C03656=1201.315,301.824,-68.864,-176.578,7.338,148.389
C03657=1201.311,302.072,-68.893,-176.576,7.341,148.389
C03658=1201.307,302.320,-68.924,-176.573,7.344,148.389
C03659=1201.303,302.568,-68.953,-176.571,7.347,148.389
C03660=1201.298,302.817,-68.983,-176.568,7.350,148.389
C03661=1201.294,303.064,-69.013,-176.566,7.352,148.389
C03662=1201.290,303.313,-69.043,-176.563,7.355,148.389
C03663=1201.285,303.561,-69.073,-176.561,7.358,148.389
C03664=1201.281,303.809,-69.103,-176.559,7.360,148.388
C03665=1201.277,304.057,-69.132,-176.556,7.363,148.388
C03666=1201.272,304.306,-69.162,-176.554,7.366,148.389
C03667=1201.268,304.553,-69.193,-176.551,7.369,148.389
C03668=1201.264,304.802,-69.222,-176.549,7.372,148.389
C03669=1201.260,305.050,-69.253,-176.546,7.375,148.389
C03670=1201.255,305.299,-69.283,-176.544,7.377,148.389
C03671=1201.251,305.547,-69.313,-176.541,7.380,148.389
C03672=1201.247,305.795,-69.343,-176.539,7.382,148.388
C03673=1201.243,306.042,-69.373,-176.536,7.385,148.388
C03674=1201.238,306.291,-69.403,-176.534,7.388,148.388
C03675=1201.234,306.539,-69.433,-176.532,7.390,148.388
C03676=1201.229,306.787,-69.463,-176.529,7.393,148.388
C03677=1201.225,307.035,-69.493,-176.527,7.397,148.389
C03678=1201.220,307.283,-69.524,-176.525,7.399,148.388
C03679=1201.217,307.532,-69.554,-176.522,7.402,148.388
C03680=1201.213,307.780,-69.584,-176.519,7.405,148.388
C03681=1201.208,308.028,-69.614,-176.517,7.407,148.388
C03682=1201.204,308.276,-69.644,-176.514,7.410,148.388
C03683=1201.199,308.524,-69.675,-176.512,7.413,148.388
C03684=1201.196,308.772,-69.705,-176.510,7.416,148.389
C03685=1201.191,309.020,-69.735,-176.507,7.419,148.389
C03686=1201.187,309.269,-69.765,-176.505,7.422,148.389
C03687=1201.183,309.517,-69.796,-176.502,7.424,148.388
C03688=1201.179,309.764,-69.826,-176.500,7.427,148.388
C03689=1201.174,310.013,-69.856,-176.497,7.430,148.388
C03690=1201.170,310.261,-69.886,-176.495,7.432,148.388
C03691=1201.165,310.509,-69.917,-176.493,7.435,148.389
C03692=1201.161,310.758,-69.948,-176.490,7.439,148.389
C03693=1201.157,311.006,-69.978,-176.488,7.441,148.389
C03694=1201.153,311.253,-70.009,-176.485,7.444,148.389
C03695=1201.149,311.501,-70.039,-176.483,7.447,148.389
C03696=1201.144,311.749,-70.069,-176.481,7.449,148.389
C03697=1201.141,311.998,-70.099,-176.478,7.452,148.389
C03698=1201.136,312.246,-70.130,-176.475,7.455,148.389
C03699=1201.131,312.494,-70.161,-176.473,7.457,148.389
C03700=1201.127,312.742,-70.191,-176.471,7.461,148.389
C03701=1201.123,312.990,-70.222,-176.468,7.464,148.389
C03702=1201.119,313.239,-70.252,-176.466,7.466,148.389
C03703=1201.115,313.487,-70.282,-176.464,7.469,148.389
C03704=1201.110,313.734,-70.313,-176.461,7.472,148.389
C03705=1201.105,313.982,-70.344,-176.459,7.474,148.389
C03706=1201.102,314.231,-70.374,-176.457,7.478,148.389
C03707=1201.097,314.507,-70.409,-176.454,7.481,148.389
C03708=1201.092,314.783,-70.442,-176.451,7.484,148.389
C03709=1201.088,315.059,-70.476,-176.448,7.487,148.389
C03710=1201.083,315.335,-70.511,-176.446,7.490,148.389
C03711=1201.078,315.584,-70.541,-176.444,7.493,148.389
C03712=1201.074,315.832,-70.572,-176.441,7.496,148.389
C03713=1201.071,316.080,-70.602,-176.439,7.498,148.389
C03714=1201.066,316.328,-70.633,-176.436,7.501,148.389
C03715=1201.062,316.575,-70.665,-176.434,7.505,148.389
C03716=1201.058,316.824,-70.696,-176.432,7.507,148.389
C03717=1201.054,317.072,-70.726,-176.429,7.510,148.389
C03718=1201.049,317.320,-70.757,-176.426,7.513,148.389
C03719=1201.044,317.568,-70.788,-176.425,7.515,148.389
C03720=1201.040,317.816,-70.819,-176.422,7.518,148.389
C03721=1201.037,318.064,-70.849,-176.419,7.521,148.389
C03722=1201.032,318.312,-70.880,-176.417,7.525,148.390
C03723=1201.028,318.561,-70.911,-176.415,7.527,148.389
C03724=1201.023,318.809,-70.942,-176.412,7.530,148.389
C03725=1201.019,319.057,-70.972,-176.410,7.533,148.390
C03726=1201.016,319.304,-71.004,-176.408,7.536,148.390
C03727=1201.011,319.552,-71.034,-176.405,7.539,148.390
C03728=1201.007,319.801,-71.065,-176.403,7.542,148.390
C03729=1201.003,320.049,-71.096,-176.401,7.544,148.390
C03730=1200.998,320.297,-71.127,-176.398,7.547,148.390
C03731=1200.994,320.545,-71.159,-176.396,7.550,148.390
C03732=1200.990,320.792,-71.189,-176.394,7.553,148.390
C03733=1200.986,321.040,-71.220,-176.391,7.556,148.390
C03734=1200.982,321.289,-71.251,-176.389,7.559,148.390
C03735=1200.977,321.536,-71.282,-176.387,7.561,148.390
C03736=1200.973,321.785,-71.313,-176.385,7.565,148.390
C03737=1200.969,322.033,-71.344,-176.382,7.568,148.390
C03738=1200.964,322.280,-71.376,-176.379,7.571,148.390
C03739=1200.960,322.529,-71.407,-176.378,7.573,148.390
C03740=1200.956,322.777,-71.438,-176.375,7.576,148.390
C03741=1200.952,323.025,-71.469,-176.372,7.579,148.390
C03742=1200.948,323.273,-71.500,-176.370,7.582,148.391
C03743=1200.944,323.522,-71.531,-176.368,7.585,148.391
C03744=1200.940,323.769,-71.562,-176.366,7.588,148.391
C03745=1200.935,324.017,-71.593,-176.363,7.590,148.391
C03746=1200.932,324.265,-71.625,-176.361,7.594,148.391
C03747=1200.927,324.513,-71.656,-176.359,7.597,148.391
C03748=1200.923,324.761,-71.687,-176.356,7.600,148.391
C03749=1200.919,325.009,-71.718,-176.354,7.602,148.391
C03750=1200.915,325.257,-71.749,-176.351,7.605,148.391
C03751=1200.910,325.505,-71.781,-176.349,7.608,148.391
C03752=1200.906,325.753,-71.812,-176.347,7.611,148.391
C03753=1200.902,326.001,-71.843,-176.345,7.614,148.392
C03754=1200.897,326.250,-71.875,-176.342,7.617,148.392
C03755=1200.893,326.497,-71.907,-176.341,7.620,148.392
C03756=1200.889,326.746,-71.938,-176.338,7.623,148.392
C03757=1200.885,326.993,-71.969,-176.336,7.626,148.392
C03758=1200.881,327.242,-72.000,-176.333,7.629,148.392
C03759=1200.876,327.489,-72.032,-176.331,7.631,148.392
C03760=1200.873,327.737,-72.064,-176.329,7.634,148.392
C03761=1200.868,327.985,-72.094,-176.326,7.638,148.392
C03762=1200.864,328.233,-72.126,-176.324,7.640,148.392
C03763=1200.860,328.481,-72.157,-176.322,7.643,148.392
C03764=1200.856,328.729,-72.189,-176.319,7.646,148.392
C03765=1200.851,328.977,-72.221,-176.318,7.649,148.393
C03766=1200.847,329.225,-72.252,-176.315,7.652,148.393
C03767=1200.843,329.473,-72.284,-176.313,7.655,148.393
C03768=1200.839,329.721,-72.315,-176.310,7.658,148.393
C03769=1200.835,329.969,-72.347,-176.308,7.661,148.393
C03770=1200.831,330.217,-72.378,-176.306,7.664,148.393
C03771=1200.826,330.465,-72.410,-176.303,7.667,148.393
C03772=1200.822,330.712,-72.442,-176.302,7.670,148.393
C03773=1200.818,330.961,-72.473,-176.299,7.673,148.393
C03774=1200.814,331.208,-72.505,-176.297,7.676,148.394
C03775=1200.810,331.456,-72.536,-176.294,7.679,148.394
C03776=1200.805,331.704,-72.569,-176.293,7.682,148.394
C03777=1200.801,331.953,-72.600,-176.290,7.685,148.394
C03778=1200.797,332.201,-72.631,-176.288,7.688,148.394
C03779=1200.793,332.448,-72.663,-176.286,7.690,148.394
C03780=1200.789,332.696,-72.695,-176.283,7.693,148.394
C03781=1200.784,332.944,-72.727,-176.281,7.697,148.394
C03782=1200.780,333.192,-72.758,-176.279,7.699,148.395
C03783=1200.776,333.440,-72.790,-176.277,7.702,148.395
C03784=1200.771,333.688,-72.822,-176.275,7.706,148.395
C03785=1200.768,333.936,-72.854,-176.272,7.709,148.395
C03786=1200.764,334.184,-72.886,-176.270,7.711,148.395
C03787=1200.760,334.431,-72.917,-176.268,7.714,148.395
C03788=1200.755,334.680,-72.950,-176.266,7.718,148.395
C03789=1200.751,334.928,-72.981,-176.264,7.720,148.395
C03790=1200.747,335.175,-73.013,-176.261,7.723,148.396
C03791=1200.743,335.424,-73.045,-176.259,7.727,148.396
C03792=1200.738,335.671,-73.077,-176.257,7.729,148.396
C03793=1200.735,335.919,-73.109,-176.255,7.732,148.396
C03794=1200.730,336.167,-73.141,-176.253,7.736,148.396
C03795=1200.726,336.415,-73.173,-176.250,7.739,148.396
C03796=1200.721,336.663,-73.205,-176.248,7.741,148.396
C03797=1200.718,336.911,-73.237,-176.246,7.744,148.397
C03798=1200.714,337.159,-73.269,-176.244,7.748,148.397
C03799=1200.709,337.407,-73.301,-176.242,7.750,148.397
C03800=1200.705,337.655,-73.333,-176.239,7.753,148.397
C03801=1200.702,337.903,-73.364,-176.237,7.757,148.397
C03802=1200.697,338.150,-73.397,-176.235,7.760,148.397
C03803=1200.693,338.398,-73.428,-176.233,7.762,148.397
C03804=1200.688,338.647,-73.461,-176.231,7.766,148.398
C03805=1200.684,338.894,-73.492,-176.228,7.769,148.398
C03806=1200.680,339.142,-73.525,-176.227,7.771,148.398
C03807=1200.676,339.390,-73.557,-176.224,7.775,148.398
C03808=1200.672,339.638,-73.590,-176.222,7.778,148.398
C03809=1200.667,339.886,-73.621,-176.220,7.780,148.398
C03810=1200.663,340.134,-73.654,-176.218,7.784,148.399
C03811=1200.659,340.412,-73.690,-176.216,7.787,148.399
C03812=1200.654,340.690,-73.726,-176.213,7.790,148.399
C03813=1200.650,340.969,-73.762,-176.210,7.794,148.399
C03814=1200.645,341.248,-73.798,-176.208,7.797,148.399
C03815=1200.640,341.495,-73.831,-176.206,7.800,148.400
C03816=1200.637,341.743,-73.863,-176.204,7.803,148.400
C03817=1200.632,341.991,-73.895,-176.202,7.807,148.400
C03818=1200.628,342.239,-73.927,-176.200,7.810,148.400
C03819=1200.624,342.486,-73.960,-176.198,7.812,148.400
C03820=1200.620,342.734,-73.992,-176.196,7.816,148.401
C03821=1200.616,342.983,-74.024,-176.194,7.819,148.401
C03822=1200.611,343.230,-74.057,-176.191,7.821,148.401
C03823=1200.608,343.478,-74.089,-176.189,7.825,148.401
C03824=1200.603,343.726,-74.121,-176.187,7.828,148.401
C03825=1200.599,343.973,-74.154,-176.185,7.831,148.401
C03826=1200.595,344.222,-74.186,-176.183,7.834,148.402
C03827=1200.591,344.470,-74.219,-176.181,7.837,148.402
C03828=1200.587,344.718,-74.251,-176.179,7.841,148.402
C03829=1200.582,344.965,-74.283,-176.177,7.843,148.402
C03830=1200.579,345.213,-74.316,-176.175,7.846,148.402
C03831=1200.574,345.461,-74.348,-176.173,7.850,148.403
C03832=1200.570,345.709,-74.382,-176.171,7.852,148.403
C03833=1200.566,345.957,-74.413,-176.169,7.856,148.403
C03834=1200.562,346.205,-74.447,-176.166,7.859,148.403
C03835=1200.557,346.452,-74.479,-176.165,7.861,148.403
C03836=1200.553,346.700,-74.512,-176.163,7.865,148.404
C03837=1200.549,346.948,-74.544,-176.160,7.868,148.404
C03838=1200.545,347.196,-74.577,-176.159,7.871,148.404
C03839=1200.541,347.444,-74.609,-176.156,7.874,148.404
C03840=1200.537,347.691,-74.642,-176.154,7.877,148.405
C03841=1200.533,347.940,-74.674,-176.152,7.881,148.405
C03842=1200.529,348.188,-74.707,-176.150,7.883,148.405
C03843=1200.524,348.435,-74.740,-176.148,7.886,148.405
C03844=1200.520,348.683,-74.772,-176.146,7.890,148.405
C03845=1200.516,348.930,-74.805,-176.145,7.893,148.406
C03846=1200.512,349.179,-74.838,-176.142,7.896,148.406
C03847=1200.507,349.426,-74.871,-176.140,7.899,148.406
C03848=1200.504,349.674,-74.903,-176.138,7.902,148.406
C03849=1200.500,349.922,-74.936,-176.136,7.905,148.407
C03850=1200.495,350.170,-74.969,-176.134,7.908,148.407
C03851=1200.491,350.418,-75.002,-176.132,7.911,148.407
C03852=1200.487,350.666,-75.035,-176.130,7.914,148.407
C03853=1200.483,350.913,-75.067,-176.128,7.918,148.408
C03854=1200.479,351.160,-75.100,-176.127,7.920,148.408
C03855=1200.475,351.408,-75.133,-176.124,7.924,148.408
C03856=1200.470,351.656,-75.165,-176.122,7.927,148.408
C03857=1200.466,351.904,-75.199,-176.121,7.930,148.409
C03858=1200.462,352.152,-75.232,-176.119,7.933,148.409
C03859=1200.459,352.399,-75.264,-176.117,7.937,148.409
C03860=1200.454,352.648,-75.297,-176.115,7.939,148.409
C03861=1200.450,352.895,-75.330,-176.113,7.942,148.410
C03862=1200.446,353.143,-75.363,-176.110,7.946,148.410
C03863=1200.442,353.391,-75.396,-176.109,7.949,148.410
C03864=1200.438,353.639,-75.429,-176.107,7.952,148.410
C03865=1200.433,353.886,-75.463,-176.105,7.955,148.411
C03866=1200.429,354.135,-75.495,-176.103,7.958,148.411
C03867=1200.426,354.382,-75.528,-176.101,7.961,148.411
C03868=1200.421,354.630,-75.561,-176.099,7.965,148.411
C03869=1200.417,354.878,-75.594,-176.097,7.967,148.412
C03870=1200.413,355.125,-75.627,-176.096,7.971,148.412
C03871=1200.409,355.373,-75.660,-176.093,7.974,148.412
C03872=1200.405,355.621,-75.693,-176.092,7.977,148.412
C03873=1200.401,355.868,-75.726,-176.090,7.980,148.413
C03874=1200.397,356.116,-75.760,-176.088,7.984,148.413
C03875=1200.392,356.364,-75.793,-176.086,7.986,148.413
C03876=1200.388,356.612,-75.826,-176.084,7.990,148.414
C03877=1200.384,356.859,-75.859,-176.082,7.993,148.414
C03878=1200.380,357.107,-75.892,-176.081,7.996,148.414
C03879=1200.376,357.355,-75.925,-176.079,7.999,148.415
C03880=1200.372,357.603,-75.959,-176.076,8.003,148.415
C03881=1200.368,357.851,-75.992,-176.075,8.005,148.415
C03882=1200.364,358.099,-76.025,-176.073,8.009,148.415
C03883=1200.360,358.346,-76.058,-176.071,8.012,148.416
C03884=1200.356,358.594,-76.092,-176.070,8.015,148.416
C03885=1200.352,358.842,-76.125,-176.068,8.019,148.417
C03886=1200.347,359.090,-76.158,-176.066,8.022,148.417
C03887=1200.343,359.337,-76.191,-176.064,8.024,148.417
C03888=1200.339,359.585,-76.224,-176.062,8.028,148.417
C03889=1200.335,359.833,-76.257,-176.061,8.031,148.418
C03890=1200.331,360.080,-76.291,-176.059,8.034,148.418
C03891=1200.327,360.328,-76.324,-176.057,8.038,148.418
C03892=1200.322,360.576,-76.358,-176.055,8.040,148.419
C03893=1200.319,360.824,-76.392,-176.054,8.044,148.419
C03894=1200.315,361.072,-76.425,-176.051,8.047,148.419
C03895=1200.310,361.320,-76.458,-176.050,8.050,148.420
C03896=1200.307,361.567,-76.492,-176.048,8.053,148.420
C03897=1200.302,361.814,-76.525,-176.047,8.056,148.420
C03898=1200.298,362.062,-76.558,-176.045,8.060,148.421
C03899=1200.294,362.310,-76.591,-176.043,8.062,148.421
C03900=1200.290,362.557,-76.625,-176.041,8.066,148.421
C03901=1200.286,362.806,-76.659,-176.040,8.070,148.422
C03902=1200.282,363.054,-76.692,-176.038,8.072,148.422
C03903=1200.278,363.301,-76.726,-176.036,8.076,148.422
C03904=1200.274,363.548,-76.759,-176.035,8.079,148.423
C03905=1200.270,363.796,-76.793,-176.033,8.082,148.423
C03906=1200.266,364.044,-76.826,-176.032,8.085,148.423
C03907=1200.262,364.292,-76.861,-176.030,8.088,148.424
C03908=1200.258,364.540,-76.894,-176.028,8.091,148.424
C03909=1200.253,364.787,-76.927,-176.026,8.095,148.424
C03910=1200.250,365.034,-76.961,-176.025,8.097,148.425
C03911=1200.245,365.282,-76.994,-176.023,8.101,148.425
C03912=1200.241,365.531,-77.028,-176.022,8.104,148.426
C03913=1200.237,365.778,-77.062,-176.020,8.107,148.426
C03914=1200.233,366.026,-77.095,-176.019,8.110,148.426
C03915=1200.228,366.306,-77.134,-176.017,8.114,148.427
C03916=1200.224,366.587,-77.172,-176.015,8.117,148.427
C03917=1200.219,366.868,-77.209,-176.013,8.121,148.428
C03918=1200.215,367.149,-77.248,-176.012,8.124,148.428
C03919=1200.211,367.396,-77.282,-176.010,8.128,148.428
C03920=1200.207,367.644,-77.316,-176.009,8.131,148.429
C03921=1200.203,367.892,-77.350,-176.007,8.135,148.429
C03922=1200.199,368.139,-77.383,-176.006,8.137,148.430
C03923=1200.195,368.386,-77.417,-176.004,8.140,148.430
C03924=1200.190,368.634,-77.450,-176.002,8.144,148.430
C03925=1200.187,368.882,-77.485,-176.001,8.146,148.431
C03926=1200.183,369.130,-77.518,-175.999,8.150,148.431
C03927=1200.178,369.377,-77.552,-175.998,8.153,148.432
C03928=1200.174,369.625,-77.585,-175.996,8.156,148.432
C03929=1200.171,369.873,-77.620,-175.995,8.159,148.432
C03930=1200.166,370.121,-77.653,-175.994,8.162,148.433
C03931=1200.162,370.368,-77.687,-175.992,8.166,148.433
C03932=1200.157,370.615,-77.722,-175.991,8.168,148.434
C03933=1200.154,370.864,-77.755,-175.990,8.171,148.434
C03934=1200.150,371.111,-77.789,-175.988,8.175,148.435
C03935=1200.145,371.359,-77.823,-175.987,8.178,148.435
C03936=1200.141,371.606,-77.857,-175.985,8.182,148.435
C03937=1200.138,371.854,-77.891,-175.984,8.184,148.436
C03938=1200.133,372.102,-77.925,-175.983,8.187,148.436
C03939=1200.129,372.349,-77.959,-175.982,8.190,148.437
C03940=1200.125,372.597,-77.993,-175.980,8.194,148.437
C03941=1200.121,372.845,-78.027,-175.979,8.197,148.437
C03942=1200.117,373.092,-78.061,-175.977,8.199,148.438
C03943=1200.113,373.340,-78.095,-175.976,8.203,148.438
C03944=1200.109,373.588,-78.128,-175.975,8.206,148.439
C03945=1200.105,373.835,-78.163,-175.974,8.209,148.439
C03946=1200.101,374.083,-78.197,-175.972,8.212,148.440
C03947=1200.097,374.331,-78.232,-175.971,8.215,148.440
C03948=1200.093,374.578,-78.265,-175.970,8.218,148.441
C03949=1200.088,374.826,-78.299,-175.969,8.221,148.441
C03950=1200.085,375.074,-78.333,-175.967,8.225,148.441
C03951=1200.080,375.321,-78.368,-175.966,8.228,148.442
C03952=1200.076,375.569,-78.401,-175.965,8.231,148.442
C03953=1200.072,375.817,-78.436,-175.964,8.234,148.443
C03954=1200.068,376.064,-78.470,-175.962,8.236,148.443
C03955=1200.064,376.312,-78.505,-175.961,8.240,148.444
C03956=1200.061,376.559,-78.539,-175.960,8.243,148.444
C03957=1200.056,376.807,-78.573,-175.959,8.246,148.445
C03958=1200.053,377.055,-78.607,-175.958,8.249,148.445
C03959=1200.048,377.302,-78.641,-175.957,8.252,148.446
C03960=1200.044,377.550,-78.675,-175.955,8.255,148.446
C03961=1200.040,377.798,-78.710,-175.954,8.259,148.447
C03962=1200.036,378.045,-78.744,-175.953,8.261,148.447
C03963=1200.032,378.292,-78.778,-175.952,8.264,148.447
C03964=1200.029,378.540,-78.812,-175.951,8.267,148.448
C03965=1200.024,378.787,-78.847,-175.950,8.270,148.448
C03966=1200.020,379.036,-78.880,-175.949,8.273,148.449
C03967=1200.016,379.283,-78.915,-175.948,8.276,148.449
C03968=1200.011,379.531,-78.949,-175.947,8.279,148.450
C03969=1200.008,379.778,-78.983,-175.946,8.282,148.450
C03970=1200.003,380.026,-79.018,-175.945,8.285,148.451
C03971=1200.000,380.273,-79.052,-175.944,8.288,148.451
C03972=1199.996,380.521,-79.087,-175.943,8.291,148.452
C03973=1199.991,380.769,-79.121,-175.941,8.295,148.452
C03974=1199.988,381.016,-79.155,-175.940,8.298,148.453
C03975=1199.983,381.264,-79.190,-175.939,8.300,148.453
C03976=1199.980,381.512,-79.224,-175.938,8.304,148.454
C03977=1199.976,381.759,-79.258,-175.937,8.306,148.454
C03978=1199.971,382.006,-79.293,-175.936,8.309,148.455
C03979=1199.968,382.254,-79.327,-175.936,8.311,148.455
C03980=1199.963,382.502,-79.362,-175.935,8.315,148.456
C03981=1199.959,382.750,-79.396,-175.934,8.317,148.456
C03982=1199.955,382.997,-79.430,-175.933,8.320,148.457
C03983=1199.951,383.244,-79.465,-175.932,8.324,148.457
C03984=1199.947,383.492,-79.500,-175.931,8.326,148.458
C03985=1199.943,383.740,-79.533,-175.930,8.329,148.458
C03986=1199.939,383.988,-79.568,-175.929,8.333,148.459
C03987=1199.935,384.234,-79.604,-175.928,8.335,148.459
C03988=1199.932,384.482,-79.638,-175.927,8.338,148.460
C03989=1199.927,384.730,-79.672,-175.927,8.342,148.461
C03990=1199.923,384.978,-79.707,-175.926,8.344,148.461
C03991=1199.919,385.225,-79.741,-175.925,8.347,148.461
C03992=1199.915,385.473,-79.776,-175.924,8.350,148.462
C03993=1199.911,385.720,-79.810,-175.923,8.353,148.462
C03994=1199.907,385.968,-79.844,-175.922,8.356,148.463
C03995=1199.903,386.215,-79.880,-175.922,8.359,148.464
C03996=1199.899,386.462,-79.914,-175.921,8.361,148.464
C03997=1199.895,386.711,-79.949,-175.920,8.364,148.465
C03998=1199.891,386.958,-79.983,-175.919,8.367,148.465
C03999=1199.887,387.206,-80.018,-175.919,8.370,148.466
C04000=1199.882,387.453,-80.052,-175.918,8.372,148.466
C04001=1199.879,387.701,-80.088,-175.917,8.375,148.467
C04002=1199.875,387.948,-80.122,-175.916,8.378,148.467
C04003=1199.871,388.196,-80.156,-175.916,8.381,148.468
C04004=1199.866,388.443,-80.191,-175.915,8.384,148.468
C04005=1199.863,388.691,-80.226,-175.914,8.386,148.469
C04006=1199.859,388.938,-80.260,-175.913,8.389,148.469
C04007=1199.855,389.186,-80.295,-175.913,8.392,148.470
C04008=1199.850,389.434,-80.330,-175.912,8.395,148.471
C04009=1199.846,389.681,-80.365,-175.912,8.398,148.471
C04010=1199.843,389.928,-80.399,-175.911,8.400,148.471
C04011=1199.839,390.176,-80.434,-175.910,8.403,148.472
C04012=1199.834,390.424,-80.468,-175.909,8.406,148.473
C04013=1199.830,390.671,-80.504,-175.909,8.408,148.473
C04014=1199.826,390.919,-80.538,-175.908,8.412,148.474
C04015=1199.823,391.166,-80.573,-175.908,8.414,148.474
C04016=1199.818,391.413,-80.608,-175.907,8.417,148.475
C04017=1199.814,391.661,-80.643,-175.907,8.419,148.475
C04018=1199.810,391.909,-80.677,-175.906,8.422,148.476
C04019=1199.806,392.192,-80.717,-175.905,8.425,148.476
C04020=1199.801,392.475,-80.757,-175.904,8.428,148.477
C04021=1199.797,392.757,-80.797,-175.904,8.432,148.478
C04022=1199.792,393.040,-80.836,-175.903,8.435,148.478
C04023=1199.788,393.288,-80.871,-175.903,8.437,148.479
C04024=1199.784,393.535,-80.906,-175.902,8.440,148.479
C04025=1199.780,393.783,-80.941,-175.901,8.442,148.480
C04026=1199.776,394.031,-80.976,-175.901,8.445,148.480
C04027=1199.772,394.278,-81.011,-175.900,8.447,148.481
C04028=1199.769,394.526,-81.046,-175.900,8.450,148.481
C04029=1199.764,394.773,-81.080,-175.899,8.453,148.482
C04030=1199.760,395.021,-81.115,-175.899,8.455,148.483
C04031=1199.756,395.268,-81.150,-175.898,8.458,148.483
C04032=1199.752,395.516,-81.185,-175.898,8.460,148.484
C04033=1199.748,395.763,-81.220,-175.897,8.463,148.484
C04034=1199.744,396.011,-81.255,-175.897,8.465,148.485
C04035=1199.740,396.259,-81.290,-175.897,8.468,148.485
C04036=1199.736,396.506,-81.324,-175.896,8.471,148.486
C04037=1199.732,396.754,-81.359,-175.896,8.473,148.486
C04038=1199.728,397.000,-81.394,-175.895,8.475,148.487
C04039=1199.724,397.249,-81.429,-175.895,8.478,148.487
C04040=1199.720,397.495,-81.464,-175.894,8.481,148.488
C04041=1199.716,397.744,-81.499,-175.894,8.483,148.488
C04042=1199.712,397.991,-81.535,-175.893,8.486,148.489
C04043=1199.707,398.238,-81.569,-175.893,8.488,148.490
C04044=1199.704,398.486,-81.605,-175.893,8.491,148.490
C04045=1199.699,398.733,-81.639,-175.892,8.494,148.491
C04046=1199.696,398.981,-81.675,-175.892,8.496,148.491
C04047=1199.692,399.229,-81.710,-175.892,8.498,148.492
C04048=1199.687,399.476,-81.745,-175.891,8.501,148.492
C04049=1199.684,399.724,-81.779,-175.890,8.503,148.493
C04050=1199.680,399.970,-81.814,-175.890,8.506,148.493
C04051=1199.676,400.219,-81.849,-175.890,8.508,148.494
C04052=1199.672,400.466,-81.885,-175.889,8.511,148.494
C04053=1199.668,400.713,-81.919,-175.889,8.513,148.495
C04054=1199.664,400.961,-81.955,-175.888,8.516,148.495
C04055=1199.659,401.208,-81.989,-175.888,8.518,148.496
C04056=1199.656,401.456,-82.025,-175.888,8.520,148.496
C04057=1199.652,401.703,-82.060,-175.887,8.523,148.497
C04058=1199.647,401.951,-82.095,-175.887,8.525,148.498
C04059=1199.644,402.198,-82.130,-175.887,8.528,148.498
C04060=1199.640,402.446,-82.165,-175.887,8.530,148.499
C04061=1199.636,402.693,-82.200,-175.886,8.532,148.499
C04062=1199.632,402.941,-82.235,-175.886,8.535,148.500
C04063=1199.627,403.188,-82.270,-175.885,8.538,148.500
C04064=1199.624,403.436,-82.306,-175.885,8.540,148.501
C04065=1199.620,403.684,-82.341,-175.884,8.542,148.501
C04066=1199.615,403.931,-82.376,-175.884,8.544,148.502
C04067=1199.612,404.179,-82.411,-175.884,8.546,148.502
C04068=1199.608,404.426,-82.446,-175.884,8.549,148.503
C04069=1199.604,404.673,-82.481,-175.883,8.551,148.503
C04070=1199.600,404.921,-82.516,-175.883,8.553,148.504
C04071=1199.596,405.169,-82.552,-175.882,8.556,148.504
C04072=1199.592,405.415,-82.587,-175.882,8.559,148.505
C04073=1199.588,405.664,-82.622,-175.882,8.561,148.505
C04074=1199.584,405.911,-82.657,-175.882,8.563,148.506
C04075=1199.580,406.158,-82.692,-175.882,8.565,148.507
C04076=1199.576,406.406,-82.727,-175.881,8.568,148.507
C04077=1199.572,406.653,-82.763,-175.881,8.570,148.508
C04078=1199.568,406.900,-82.798,-175.881,8.572,148.508
C04079=1199.564,407.148,-82.833,-175.880,8.574,148.508
C04080=1199.560,407.396,-82.868,-175.880,8.576,148.509
C04081=1199.556,407.643,-82.904,-175.880,8.579,148.509
C04082=1199.552,407.891,-82.938,-175.879,8.581,148.510
C04083=1199.548,408.139,-82.975,-175.879,8.583,148.511
C04084=1199.543,408.385,-83.010,-175.879,8.585,148.511
C04085=1199.539,408.634,-83.045,-175.879,8.588,148.512
C04086=1199.536,408.881,-83.080,-175.879,8.590,148.512
C04087=1199.531,409.128,-83.115,-175.878,8.592,148.513
C04088=1199.528,409.375,-83.151,-175.878,8.595,148.513
C04089=1199.524,409.623,-83.186,-175.877,8.596,148.514
C04090=1199.520,409.870,-83.221,-175.877,8.599,148.514
C04091=1199.516,410.118,-83.256,-175.877,8.601,148.515
C04092=1199.512,410.365,-83.292,-175.877,8.603,148.515
C04093=1199.508,410.613,-83.326,-175.876,8.606,148.516
C04094=1199.504,410.860,-83.362,-175.876,8.608,148.516
C04095=1199.500,411.108,-83.398,-175.876,8.610,148.517
C04096=1199.496,411.354,-83.433,-175.876,8.612,148.517
C04097=1199.491,411.603,-83.468,-175.876,8.613,148.517
C04098=1199.488,411.850,-83.504,-175.875,8.616,148.518
C04099=1199.484,412.098,-83.539,-175.875,8.618,148.519
C04100=1199.480,412.345,-83.574,-175.875,8.620,148.519
C04101=1199.476,412.592,-83.610,-175.875,8.623,148.520
C04102=1199.472,412.840,-83.645,-175.874,8.625,148.520
C04103=1199.468,413.087,-83.680,-175.874,8.627,148.521
C04104=1199.464,413.335,-83.716,-175.874,8.629,148.521
C04105=1199.461,413.582,-83.751,-175.873,8.631,148.522
C04106=1199.456,413.829,-83.787,-175.873,8.634,148.522
C04107=1199.452,414.077,-83.822,-175.873,8.635,148.523
C04108=1199.448,414.325,-83.857,-175.873,8.637,148.523
C04109=1199.444,414.572,-83.893,-175.873,8.640,148.524
C04110=1199.440,414.819,-83.928,-175.872,8.642,148.524
C04111=1199.436,415.067,-83.964,-175.872,8.644,148.524
C04112=1199.432,415.315,-83.998,-175.872,8.646,148.525
C04113=1199.427,415.562,-84.034,-175.872,8.648,148.525
C04114=1199.424,415.809,-84.070,-175.872,8.650,148.526
C04115=1199.419,416.132,-84.116,-175.871,8.653,148.527
C04116=1199.415,416.457,-84.162,-175.871,8.655,148.527
C04117=1199.414,416.780,-84.208,-175.871,8.658,148.528
C04118=1199.417,417.103,-84.254,-175.870,8.661,148.528
C04119=1198.995,417.104,-84.292,-175.873,8.671,148.532
C04120=1198.992,416.778,-84.247,-175.874,8.669,148.532
C04121=1198.993,416.452,-84.200,-175.874,8.666,148.531
C04122=1198.997,416.125,-84.154,-175.874,8.664,148.530
C04123=1199.003,415.799,-84.107,-175.875,8.660,148.530
C04124=1199.007,415.551,-84.072,-175.875,8.659,148.529
C04125=1199.010,415.304,-84.036,-175.875,8.657,148.529
C04126=1199.015,415.056,-84.000,-175.875,8.654,148.528
C04127=1199.019,414.809,-83.965,-175.875,8.652,148.528
C04128=1199.023,414.561,-83.930,-175.876,8.650,148.527
C04129=1199.026,414.313,-83.894,-175.876,8.648,148.527
C04130=1199.030,414.066,-83.859,-175.877,8.646,148.526
C04131=1199.034,413.819,-83.824,-175.876,8.644,148.526
C04132=1199.038,413.572,-83.788,-175.877,8.642,148.525
C04133=1199.042,413.324,-83.752,-175.877,8.640,148.525
C04134=1199.047,413.076,-83.717,-175.877,8.637,148.524
C04135=1199.051,412.829,-83.682,-175.878,8.635,148.524
C04136=1199.054,412.581,-83.646,-175.878,8.633,148.523
C04137=1199.058,412.334,-83.611,-175.878,8.631,148.523
C04138=1199.062,412.087,-83.576,-175.878,8.629,148.522
C04139=1199.066,411.839,-83.541,-175.878,8.627,148.522
C04140=1199.070,411.592,-83.505,-175.878,8.625,148.521
C04141=1199.074,411.345,-83.470,-175.879,8.623,148.521
C04142=1199.078,411.097,-83.434,-175.879,8.621,148.520
C04143=1199.083,410.849,-83.399,-175.879,8.618,148.520
C04144=1199.087,410.602,-83.364,-175.880,8.616,148.519
C04145=1199.090,410.354,-83.328,-175.880,8.614,148.519
C04146=1199.094,410.107,-83.293,-175.880,8.612,148.518
C04147=1199.099,409.860,-83.258,-175.880,8.609,148.518
C04148=1199.102,409.612,-83.223,-175.881,8.607,148.517
C04149=1199.106,409.365,-83.187,-175.881,8.605,148.517
C04150=1199.110,409.117,-83.152,-175.881,8.603,148.516
C04151=1199.114,408.870,-83.117,-175.881,8.600,148.516
C04152=1199.118,408.622,-83.082,-175.882,8.598,148.515
C04153=1199.122,408.375,-83.046,-175.882,8.596,148.515
C04154=1199.126,408.128,-83.011,-175.882,8.594,148.514
C04155=1199.130,407.880,-82.976,-175.883,8.592,148.514
C04156=1199.134,407.632,-82.940,-175.883,8.589,148.513
C04157=1199.139,407.385,-82.905,-175.883,8.587,148.513
C04158=1199.142,407.137,-82.870,-175.883,8.585,148.512
C04159=1199.146,406.889,-82.834,-175.884,8.583,148.512
C04160=1199.150,406.643,-82.799,-175.884,8.580,148.511
C04161=1199.154,406.395,-82.764,-175.884,8.578,148.511
C04162=1199.158,406.147,-82.729,-175.884,8.576,148.510
C04163=1199.162,405.900,-82.694,-175.885,8.573,148.509
C04164=1199.166,405.652,-82.659,-175.885,8.571,148.509
C04165=1199.170,405.405,-82.623,-175.885,8.569,148.509
C04166=1199.174,405.158,-82.588,-175.886,8.567,148.508
C04167=1199.178,404.910,-82.553,-175.886,8.565,148.508
C04168=1199.182,404.662,-82.518,-175.886,8.562,148.507
C04169=1199.186,404.415,-82.483,-175.887,8.559,148.506
C04170=1199.190,404.167,-82.448,-175.887,8.557,148.506
C04171=1199.194,403.920,-82.412,-175.887,8.555,148.505
C04172=1199.198,403.673,-82.377,-175.888,8.553,148.505
C04173=1199.202,403.425,-82.342,-175.888,8.550,148.504
C04174=1199.206,403.178,-82.307,-175.888,8.548,148.504
C04175=1199.210,402.930,-82.272,-175.888,8.546,148.503
C04176=1199.214,402.682,-82.237,-175.889,8.543,148.503
C04177=1199.218,402.436,-82.201,-175.889,8.540,148.502
C04178=1199.222,402.188,-82.167,-175.890,8.538,148.502
C04179=1199.226,401.940,-82.131,-175.890,8.536,148.501
C04180=1199.230,401.693,-82.097,-175.890,8.534,148.501
C04181=1199.234,401.445,-82.061,-175.890,8.531,148.500
C04182=1199.238,401.198,-82.026,-175.890,8.529,148.499
C04183=1199.242,400.950,-81.991,-175.891,8.526,148.499
C04184=1199.246,400.703,-81.955,-175.892,8.524,148.499
C04185=1199.250,400.455,-81.921,-175.892,8.522,148.498
C04186=1199.254,400.208,-81.885,-175.892,8.519,148.497
C04187=1199.258,399.960,-81.851,-175.893,8.516,148.497
C04188=1199.262,399.713,-81.815,-175.893,8.514,148.496
C04189=1199.266,399.465,-81.781,-175.894,8.512,148.496
C04190=1199.271,399.218,-81.745,-175.894,8.509,148.495
C04191=1199.275,398.970,-81.711,-175.895,8.506,148.495
C04192=1199.277,398.723,-81.676,-175.895,8.504,148.494
C04193=1199.282,398.475,-81.641,-175.895,8.502,148.494
C04194=1199.286,398.228,-81.606,-175.896,8.499,148.493
C04195=1199.290,397.980,-81.571,-175.896,8.496,148.493
C04196=1199.294,397.733,-81.536,-175.896,8.494,148.492
C04197=1199.298,397.485,-81.501,-175.897,8.492,148.491
C04198=1199.302,397.238,-81.466,-175.897,8.489,148.491
C04199=1199.306,396.990,-81.431,-175.898,8.487,148.490
C04200=1199.310,396.743,-81.396,-175.898,8.483,148.490
C04201=1199.314,396.495,-81.361,-175.899,8.481,148.489
C04202=1199.319,396.248,-81.326,-175.899,8.479,148.489
C04203=1199.323,396.000,-81.291,-175.900,8.476,148.488
C04204=1199.326,395.752,-81.255,-175.900,8.474,148.488
C04205=1199.330,395.505,-81.221,-175.900,8.472,148.487
C04206=1199.334,395.257,-81.186,-175.901,8.468,148.487
C04207=1199.338,395.010,-81.151,-175.901,8.466,148.486
C04208=1199.342,394.762,-81.116,-175.902,8.463,148.486
C04209=1199.347,394.515,-81.081,-175.902,8.461,148.485
C04210=1199.351,394.267,-81.046,-175.903,8.458,148.484
C04211=1199.354,394.019,-81.012,-175.903,8.455,148.484
C04212=1199.358,393.773,-80.977,-175.904,8.452,148.483
C04213=1199.362,393.525,-80.942,-175.905,8.450,148.483
C04214=1199.366,393.278,-80.907,-175.905,8.448,148.482
C04215=1199.370,393.030,-80.872,-175.906,8.445,148.482
C04216=1199.374,392.747,-80.832,-175.906,8.442,148.481
C04217=1199.380,392.464,-80.793,-175.907,8.439,148.480
C04218=1199.384,392.182,-80.753,-175.908,8.435,148.480
C04219=1199.389,391.898,-80.713,-175.909,8.432,148.479
C04220=1199.393,391.651,-80.679,-175.909,8.430,148.479
C04221=1199.396,391.403,-80.643,-175.910,8.427,148.478
C04222=1199.401,391.156,-80.609,-175.910,8.425,148.478
C04223=1199.405,390.908,-80.574,-175.911,8.422,148.477
C04224=1199.409,390.661,-80.539,-175.911,8.420,148.477
C04225=1199.412,390.413,-80.505,-175.912,8.417,148.476
C04226=1199.417,390.166,-80.470,-175.913,8.413,148.476
C04227=1199.421,389.918,-80.435,-175.913,8.411,148.475
C04228=1199.425,389.671,-80.400,-175.914,8.408,148.474
C04229=1199.429,389.422,-80.365,-175.915,8.405,148.474
C04230=1199.433,389.175,-80.331,-175.915,8.403,148.473
C04231=1199.437,388.928,-80.296,-175.916,8.400,148.473
C04232=1199.441,388.680,-80.261,-175.917,8.397,148.472
C04233=1199.445,388.432,-80.227,-175.917,8.394,148.472
C04234=1199.449,388.185,-80.193,-175.918,8.391,148.471
C04235=1199.453,387.938,-80.157,-175.919,8.389,148.471
C04236=1199.457,387.690,-80.123,-175.919,8.386,148.470
C04237=1199.461,387.442,-80.088,-175.920,8.383,148.470
C04238=1199.465,387.195,-80.054,-175.921,8.380,148.469
C04239=1199.469,386.947,-80.019,-175.922,8.377,148.469
C04240=1199.473,386.700,-79.984,-175.922,8.375,148.468
C04241=1199.477,386.452,-79.949,-175.923,8.372,148.468
C04242=1199.481,386.205,-79.915,-175.924,8.369,148.467
C04243=1199.485,385.957,-79.880,-175.925,8.366,148.467
C04244=1199.490,385.709,-79.846,-175.926,8.363,148.466
C04245=1199.494,385.461,-79.811,-175.926,8.361,148.465
C04246=1199.497,385.215,-79.777,-175.927,8.358,148.465
C04247=1199.501,384.967,-79.742,-175.928,8.355,148.464
C04248=1199.506,384.719,-79.707,-175.929,8.352,148.464
C04249=1199.509,384.471,-79.673,-175.930,8.349,148.463
C04250=1199.513,384.224,-79.639,-175.931,8.346,148.463
C04251=1199.517,383.976,-79.604,-175.932,8.343,148.462
C04252=1199.521,383.729,-79.570,-175.932,8.340,148.462
C04253=1199.526,383.481,-79.535,-175.933,8.338,148.461
C04254=1199.530,383.233,-79.501,-175.934,8.334,148.461
C04255=1199.533,382.987,-79.466,-175.935,8.332,148.460
C04256=1199.537,382.739,-79.431,-175.936,8.329,148.460
C04257=1199.542,382.491,-79.397,-175.937,8.325,148.459
C04258=1199.545,382.243,-79.362,-175.938,8.323,148.459
C04259=1199.550,381.996,-79.328,-175.939,8.320,148.458
C04260=1199.554,381.749,-79.293,-175.940,8.317,148.458
C04261=1199.557,381.501,-79.259,-175.941,8.314,148.457
C04262=1199.562,381.253,-79.225,-175.941,8.311,148.457
C04263=1199.566,381.005,-79.190,-175.943,8.308,148.456
C04264=1199.570,380.758,-79.156,-175.943,8.305,148.456
C04265=1199.574,380.510,-79.121,-175.945,8.302,148.455
C04266=1199.578,380.263,-79.087,-175.945,8.299,148.455
C04267=1199.582,380.015,-79.053,-175.947,8.296,148.454
C04268=1199.586,379.767,-79.018,-175.947,8.293,148.454
C04269=1199.590,379.520,-78.984,-175.949,8.290,148.453
C04270=1199.594,379.272,-78.949,-175.950,8.286,148.453
C04271=1199.598,379.025,-78.916,-175.951,8.283,148.452
C04272=1199.603,378.777,-78.882,-175.952,8.280,148.452
C04273=1199.607,378.529,-78.847,-175.953,8.277,148.451
C04274=1199.610,378.282,-78.813,-175.954,8.275,148.451
C04275=1199.615,378.034,-78.779,-175.955,8.271,148.450
C04276=1199.618,377.786,-78.744,-175.956,8.269,148.450
C04277=1199.623,377.539,-78.710,-175.958,8.266,148.450
C04278=1199.626,377.291,-78.676,-175.958,8.263,148.449
C04279=1199.631,377.044,-78.641,-175.960,8.259,148.449
C04280=1199.634,376.797,-78.607,-175.961,8.256,148.448
C04281=1199.639,376.548,-78.573,-175.962,8.253,148.448
C04282=1199.643,376.301,-78.539,-175.963,8.250,148.447
C04283=1199.647,376.053,-78.505,-175.964,8.247,148.447
C04284=1199.650,375.806,-78.471,-175.966,8.244,148.446
C04285=1199.655,375.558,-78.436,-175.967,8.241,148.446
C04286=1199.659,375.311,-78.403,-175.968,8.238,148.445
C04287=1199.663,375.062,-78.368,-175.969,8.235,148.445
C04288=1199.667,374.815,-78.334,-175.971,8.231,148.444
C04289=1199.671,374.568,-78.300,-175.972,8.228,148.444
C04290=1199.675,374.320,-78.266,-175.973,8.226,148.444
C04291=1199.680,374.072,-78.232,-175.974,8.223,148.443
C04292=1199.683,373.825,-78.198,-175.976,8.219,148.443
C04293=1199.687,373.577,-78.163,-175.977,8.216,148.442
C04294=1199.691,373.330,-78.129,-175.978,8.213,148.442
C04295=1199.695,373.082,-78.096,-175.980,8.211,148.441
C04296=1199.699,372.834,-78.061,-175.981,8.207,148.441
C04297=1199.703,372.587,-78.027,-175.982,8.204,148.440
C04298=1199.708,372.339,-77.994,-175.983,8.201,148.440
C04299=1199.712,372.092,-77.960,-175.985,8.197,148.440
C04300=1199.716,371.843,-77.925,-175.986,8.195,148.439
C04301=1199.720,371.596,-77.892,-175.988,8.192,148.439
C04302=1199.724,371.349,-77.858,-175.989,8.188,148.438
C04303=1199.728,371.100,-77.823,-175.991,8.185,148.438
C04304=1199.732,370.853,-77.790,-175.992,8.182,148.438
C04305=1199.736,370.606,-77.756,-175.994,8.179,148.437
C04306=1199.741,370.358,-77.722,-175.994,8.176,148.437
C04307=1199.744,370.110,-77.688,-175.996,8.172,148.436
C04308=1199.748,369.862,-77.654,-175.997,8.169,148.436
C04309=1199.753,369.615,-77.620,-175.999,8.166,148.435
C04310=1199.756,369.368,-77.587,-176.000,8.163,148.435
C04311=1199.761,369.119,-77.552,-176.002,8.160,148.434
C04312=1199.764,368.872,-77.519,-176.003,8.156,148.434
C04313=1199.769,368.624,-77.485,-176.005,8.154,148.434
C04314=1199.773,368.377,-77.451,-176.007,8.150,148.433
C04315=1199.777,368.128,-77.417,-176.008,8.147,148.433
C04316=1199.781,367.881,-77.384,-176.009,8.145,148.433
C04317=1199.785,367.633,-77.350,-176.011,8.141,148.432
C04318=1199.789,367.386,-77.316,-176.012,8.138,148.432
C04319=1199.793,367.137,-77.282,-176.014,8.135,148.431
C04320=1199.798,366.857,-77.244,-176.016,8.131,148.431
C04321=1199.802,366.576,-77.205,-176.018,8.127,148.430
C04322=1199.806,366.296,-77.168,-176.019,8.124,148.430
C04323=1199.811,366.015,-77.130,-176.021,8.120,148.430
C04324=1199.815,365.768,-77.096,-176.022,8.117,148.429
C04325=1199.820,365.520,-77.062,-176.025,8.114,148.429
C04326=1199.824,365.272,-77.028,-176.026,8.111,148.429
C04327=1199.827,365.024,-76.995,-176.028,8.107,148.428
C04328=1199.832,364.776,-76.962,-176.029,8.105,148.428
C04329=1199.835,364.529,-76.928,-176.031,8.101,148.427
C04330=1199.840,364.281,-76.894,-176.032,8.098,148.427
C04331=1199.844,364.033,-76.861,-176.034,8.095,148.427
C04332=1199.848,363.786,-76.827,-176.035,8.092,148.426
C04333=1199.852,363.538,-76.793,-176.037,8.089,148.426
C04334=1199.856,363.290,-76.760,-176.039,8.086,148.426
C04335=1199.860,363.043,-76.726,-176.040,8.082,148.425
C04336=1199.865,362.795,-76.693,-176.043,8.079,148.425
C04337=1199.869,362.547,-76.660,-176.044,8.076,148.425
C04338=1199.873,362.300,-76.626,-176.046,8.072,148.424
C04339=1199.876,362.052,-76.592,-176.047,8.070,148.424
C04340=1199.880,361.804,-76.559,-176.049,8.066,148.424
C04341=1199.884,361.556,-76.526,-176.051,8.063,148.423
C04342=1199.889,361.308,-76.492,-176.053,8.060,148.423
C04343=1199.893,361.061,-76.458,-176.054,8.057,148.423
C04344=1199.897,360.813,-76.425,-176.056,8.054,148.422
C04345=1199.901,360.566,-76.392,-176.058,8.050,148.422
C04346=1199.905,360.318,-76.359,-176.060,8.047,148.422
C04347=1199.909,360.069,-76.325,-176.061,8.044,148.421
C04348=1199.913,359.822,-76.292,-176.063,8.041,148.421
C04349=1199.917,359.575,-76.258,-176.065,8.038,148.421
C04350=1199.921,359.327,-76.225,-176.066,8.034,148.420
C04351=1199.925,359.079,-76.192,-176.069,8.031,148.420
C04352=1199.929,358.831,-76.159,-176.070,8.028,148.420
C04353=1199.934,358.584,-76.126,-176.072,8.025,148.419
C04354=1199.938,358.336,-76.092,-176.074,8.022,148.419
C04355=1199.942,358.088,-76.059,-176.076,8.019,148.419
C04356=1199.946,357.841,-76.026,-176.078,8.016,148.419
C04357=1199.950,357.593,-75.993,-176.080,8.012,148.418
C04358=1199.954,357.345,-75.960,-176.081,8.009,148.418
C04359=1199.958,357.097,-75.926,-176.083,8.006,148.418
C04360=1199.962,356.849,-75.893,-176.085,8.002,148.417
C04361=1199.966,356.601,-75.860,-176.087,8.000,148.417
C04362=1199.970,356.353,-75.827,-176.089,7.996,148.417
C04363=1199.974,356.106,-75.794,-176.091,7.993,148.416
C04364=1199.978,355.858,-75.760,-176.093,7.990,148.416
C04365=1199.983,355.610,-75.727,-176.094,7.987,148.416
C04366=1199.987,355.363,-75.694,-176.097,7.983,148.416
C04367=1199.991,355.115,-75.661,-176.098,7.981,148.415
C04368=1199.995,354.867,-75.628,-176.100,7.977,148.415
C04369=1199.999,354.619,-75.595,-176.102,7.974,148.415
C04370=1200.003,354.372,-75.562,-176.104,7.971,148.415
C04371=1200.007,354.124,-75.528,-176.106,7.968,148.414
C04372=1200.012,353.876,-75.495,-176.108,7.964,148.414
C04373=1200.016,353.628,-75.463,-176.110,7.962,148.414
C04374=1200.020,353.380,-75.430,-176.112,7.959,148.414
C04375=1200.024,353.132,-75.396,-176.114,7.955,148.413
C04376=1200.028,352.885,-75.364,-176.115,7.953,148.413
C04377=1200.032,352.637,-75.331,-176.117,7.949,148.413
C04378=1200.036,352.389,-75.298,-176.120,7.946,148.412
C04379=1200.040,352.141,-75.265,-176.121,7.943,148.412
C04380=1200.045,351.893,-75.232,-176.123,7.940,148.412
C04381=1200.049,351.646,-75.199,-176.125,7.936,148.412
C04382=1200.053,351.398,-75.166,-176.127,7.934,148.411
C04383=1200.057,351.150,-75.134,-176.129,7.931,148.411
C04384=1200.061,350.903,-75.101,-176.131,7.927,148.411
C04385=1200.065,350.655,-75.068,-176.133,7.924,148.411
C04386=1200.070,350.407,-75.035,-176.135,7.921,148.410
C04387=1200.074,350.159,-75.002,-176.137,7.918,148.410
C04388=1200.077,349.912,-74.970,-176.139,7.914,148.410
C04389=1200.082,349.664,-74.937,-176.141,7.912,148.410
C04390=1200.086,349.416,-74.904,-176.143,7.909,148.410
C04391=1200.090,349.168,-74.871,-176.145,7.905,148.409
C04392=1200.095,348.919,-74.839,-176.147,7.902,148.409
C04393=1200.098,348.672,-74.806,-176.149,7.899,148.409
C04394=1200.102,348.424,-74.773,-176.151,7.896,148.408
C04395=1200.107,348.176,-74.740,-176.153,7.893,148.408
C04396=1200.111,347.929,-74.708,-176.155,7.890,148.408
C04397=1200.115,347.681,-74.676,-176.157,7.887,148.408
C04398=1200.119,347.433,-74.643,-176.159,7.883,148.408
C04399=1200.123,347.185,-74.609,-176.161,7.881,148.407
C04400=1200.127,346.937,-74.578,-176.163,7.877,148.407
C04401=1200.131,346.690,-74.544,-176.166,7.874,148.407
C04402=1200.136,346.441,-74.512,-176.167,7.872,148.407
C04403=1200.140,346.194,-74.479,-176.169,7.868,148.407
C04404=1200.144,345.946,-74.447,-176.172,7.865,148.406
C04405=1200.148,345.699,-74.414,-176.173,7.862,148.406
C04406=1200.153,345.450,-74.382,-176.176,7.859,148.406
C04407=1200.156,345.203,-74.349,-176.178,7.856,148.406
C04408=1200.160,344.954,-74.317,-176.179,7.853,148.406
C04409=1200.165,344.707,-74.285,-176.182,7.850,148.405
C04410=1200.169,344.459,-74.252,-176.184,7.846,148.405
C04411=1200.173,344.211,-74.220,-176.186,7.843,148.405
C04412=1200.177,343.964,-74.187,-176.188,7.841,148.405
C04413=1200.181,343.715,-74.155,-176.190,7.837,148.405
C04414=1200.186,343.467,-74.122,-176.192,7.834,148.404
C04415=1200.190,343.220,-74.090,-176.194,7.831,148.404
C04416=1200.194,342.972,-74.058,-176.196,7.828,148.404
C04417=1200.198,342.724,-74.026,-176.198,7.825,148.404
C04418=1200.202,342.476,-73.993,-176.201,7.822,148.404
C04419=1200.207,342.228,-73.961,-176.203,7.819,148.403
C04420=1200.211,341.980,-73.929,-176.205,7.816,148.403
C04421=1200.215,341.733,-73.896,-176.207,7.813,148.403
C04422=1200.218,341.485,-73.864,-176.209,7.810,148.403
C04423=1200.223,341.236,-73.831,-176.211,7.807,148.403
C04424=1200.228,340.958,-73.795,-176.213,7.803,148.402
C04425=1200.232,340.680,-73.758,-176.216,7.800,148.402
C04426=1200.237,340.402,-73.723,-176.219,7.796,148.402
C04427=1200.242,340.123,-73.687,-176.221,7.793,148.402
C04428=1200.246,339.875,-73.655,-176.223,7.790,148.402
C04429=1200.249,339.627,-73.622,-176.225,7.787,148.402
C04430=1200.254,339.380,-73.590,-176.228,7.784,148.402
C04431=1200.258,339.132,-73.558,-176.230,7.781,148.401
C04432=1200.263,338.883,-73.526,-176.231,7.778,148.401
C04433=1200.267,338.636,-73.494,-176.234,7.775,148.401
C04434=1200.271,338.388,-73.462,-176.236,7.771,148.401
C04435=1200.275,338.140,-73.429,-176.238,7.769,148.401
C04436=1200.278,337.892,-73.397,-176.240,7.766,148.401
C04437=1200.283,337.645,-73.365,-176.243,7.763,148.400
C04438=1200.287,337.396,-73.333,-176.245,7.759,148.400
C04439=1200.292,337.148,-73.301,-176.247,7.757,148.400
C04440=1200.296,336.901,-73.269,-176.249,7.754,148.400
C04441=1200.300,336.653,-73.238,-176.251,7.750,148.400
C04442=1200.304,336.404,-73.205,-176.253,7.748,148.400
C04443=1200.308,336.157,-73.174,-176.256,7.745,148.400
C04444=1200.312,335.909,-73.142,-176.258,7.742,148.399
C04445=1200.317,335.661,-73.109,-176.260,7.739,148.399
C04446=1200.321,335.413,-73.078,-176.262,7.736,148.399
C04447=1200.325,335.165,-73.046,-176.264,7.733,148.399
C04448=1200.329,334.917,-73.014,-176.267,7.729,148.399
C04449=1200.333,334.670,-72.982,-176.268,7.727,148.399
C04450=1200.337,334.422,-72.950,-176.271,7.724,148.398
C04451=1200.341,334.173,-72.918,-176.273,7.720,148.398
C04452=1200.346,333.926,-72.886,-176.275,7.718,148.398
C04453=1200.349,333.678,-72.855,-176.278,7.715,148.398
C04454=1200.354,333.429,-72.823,-176.280,7.712,148.398
C04455=1200.359,333.182,-72.791,-176.283,7.709,148.398
C04456=1200.362,332.934,-72.760,-176.284,7.706,148.398
C04457=1200.367,332.686,-72.728,-176.286,7.703,148.397
C04458=1200.371,332.438,-72.696,-176.289,7.700,148.397
C04459=1200.375,332.190,-72.664,-176.291,7.697,148.397
C04460=1200.379,331.942,-72.633,-176.293,7.694,148.397
C04461=1200.383,331.694,-72.601,-176.296,7.691,148.397
C04462=1200.388,331.446,-72.569,-176.298,7.687,148.397
C04463=1200.392,331.198,-72.537,-176.300,7.685,148.397
C04464=1200.395,330.950,-72.505,-176.302,7.682,148.397
C04465=1200.400,330.702,-72.475,-176.304,7.679,148.396
C04466=1200.405,330.454,-72.442,-176.307,7.676,148.397
C04467=1200.409,330.206,-72.411,-176.309,7.673,148.396
C04468=1200.413,329.958,-72.380,-176.312,7.670,148.396
C04469=1200.417,329.710,-72.348,-176.314,7.667,148.396
C04470=1200.421,329.462,-72.316,-176.316,7.665,148.396
C04471=1200.425,329.215,-72.285,-176.318,7.661,148.396
C04472=1200.430,328.966,-72.253,-176.321,7.658,148.396
C04473=1200.434,328.718,-72.221,-176.322,7.656,148.396
C04474=1200.438,328.470,-72.190,-176.325,7.652,148.396
C04475=1200.442,328.222,-72.159,-176.327,7.649,148.396
C04476=1200.446,327.975,-72.127,-176.330,7.646,148.395
C04477=1200.450,327.726,-72.096,-176.332,7.644,148.395
C04478=1200.455,327.479,-72.065,-176.334,7.640,148.395
C04479=1200.458,327.231,-72.033,-176.337,7.637,148.395
C04480=1200.463,326.983,-72.002,-176.338,7.635,148.395
C04481=1200.467,326.735,-71.970,-176.341,7.632,148.395
C04482=1200.472,326.486,-71.939,-176.343,7.629,148.395
C04483=1200.476,326.238,-71.907,-176.345,7.626,148.395
C04484=1200.480,325.990,-71.876,-176.348,7.623,148.395
C04485=1200.484,325.742,-71.844,-176.350,7.620,148.395
C04486=1200.489,325.494,-71.813,-176.353,7.617,148.395
C04487=1200.492,325.246,-71.782,-176.355,7.614,148.394
C04488=1200.497,324.998,-71.751,-176.357,7.611,148.394
C04489=1200.501,324.751,-71.719,-176.360,7.608,148.394
C04490=1200.505,324.502,-71.688,-176.362,7.606,148.394
C04491=1200.510,324.254,-71.657,-176.364,7.603,148.394
C04492=1200.514,324.006,-71.626,-176.367,7.600,148.394
C04493=1200.518,323.758,-71.595,-176.369,7.597,148.394
C04494=1200.522,323.510,-71.563,-176.371,7.594,148.394
C04495=1200.526,323.262,-71.532,-176.374,7.591,148.394
C04496=1200.530,323.014,-71.501,-176.376,7.588,148.394
C04497=1200.534,322.767,-71.470,-176.378,7.585,148.394
C04498=1200.539,322.519,-71.439,-176.380,7.582,148.394
C04499=1200.543,322.270,-71.408,-176.383,7.579,148.394
C04500=1200.547,322.023,-71.377,-176.385,7.577,148.394
C04501=1200.551,321.774,-71.346,-176.387,7.574,148.393
C04502=1200.556,321.526,-71.315,-176.390,7.571,148.393
C04503=1200.559,321.278,-71.283,-176.393,7.568,148.393
C04504=1200.564,321.030,-71.252,-176.394,7.565,148.393
C04505=1200.569,320.782,-71.222,-176.397,7.562,148.393
C04506=1200.573,320.534,-71.190,-176.399,7.559,148.393
C04507=1200.576,320.287,-71.160,-176.401,7.556,148.393
C04508=1200.581,320.039,-71.129,-176.404,7.553,148.393
C04509=1200.585,319.790,-71.098,-176.406,7.550,148.393
C04510=1200.589,319.542,-71.067,-176.408,7.548,148.393
C04511=1200.593,319.294,-71.035,-176.411,7.545,148.393
C04512=1200.598,319.046,-71.004,-176.413,7.542,148.393
C04513=1200.602,318.798,-70.974,-176.415,7.539,148.393
C04514=1200.606,318.550,-70.943,-176.418,7.536,148.393
C04515=1200.610,318.302,-70.912,-176.420,7.533,148.393
C04516=1200.615,318.054,-70.882,-176.423,7.530,148.393
C04517=1200.619,317.805,-70.850,-176.425,7.528,148.393
C04518=1200.623,317.557,-70.820,-176.428,7.525,148.393
C04519=1200.627,317.310,-70.789,-176.430,7.521,148.392
C04520=1200.631,317.061,-70.758,-176.432,7.519,148.392
C04521=1200.636,316.814,-70.727,-176.435,7.516,148.392
C04522=1200.639,316.566,-70.697,-176.437,7.513,148.392
C04523=1200.644,316.317,-70.666,-176.439,7.511,148.392
C04524=1200.648,316.069,-70.635,-176.442,7.508,148.392
C04525=1200.653,315.821,-70.604,-176.445,7.505,148.392
C04526=1200.657,315.574,-70.574,-176.446,7.502,148.392
C04527=1200.661,315.325,-70.543,-176.449,7.499,148.392
C04528=1200.666,315.049,-70.509,-176.452,7.496,148.392
C04529=1200.670,314.773,-70.475,-176.454,7.493,148.392
C04530=1200.675,314.496,-70.440,-176.457,7.490,148.392
C04531=1200.680,314.220,-70.407,-176.460,7.486,148.392
C04532=1200.684,313.972,-70.376,-176.462,7.484,148.392
C04533=1200.688,313.724,-70.346,-176.465,7.481,148.392
C04534=1200.692,313.476,-70.315,-176.467,7.478,148.392
C04535=1200.697,313.228,-70.284,-176.469,7.475,148.392
C04536=1200.701,312.980,-70.254,-176.472,7.472,148.392
C04537=1200.705,312.732,-70.223,-176.474,7.469,148.392
C04538=1200.710,312.483,-70.192,-176.477,7.467,148.392
C04539=1200.714,312.235,-70.162,-176.479,7.464,148.392
C04540=1200.718,311.987,-70.132,-176.481,7.461,148.392
C04541=1200.722,311.740,-70.101,-176.484,7.458,148.392
C04542=1200.727,311.492,-70.071,-176.486,7.455,148.392
C04543=1200.731,311.242,-70.040,-176.489,7.452,148.392
C04544=1200.735,310.995,-70.010,-176.491,7.450,148.392
C04545=1200.739,310.747,-69.979,-176.494,7.447,148.392
C04546=1200.743,310.499,-69.949,-176.496,7.444,148.392
C04547=1200.748,310.250,-69.919,-176.498,7.442,148.392
C04548=1200.752,310.002,-69.889,-176.501,7.439,148.392
C04549=1200.756,309.754,-69.858,-176.504,7.435,148.392
C04550=1200.760,309.506,-69.828,-176.506,7.433,148.392
C04551=1200.765,309.258,-69.798,-176.508,7.430,148.392
C04552=1200.770,309.010,-69.767,-176.511,7.427,148.392
C04553=1200.774,308.762,-69.737,-176.513,7.425,148.392
C04554=1200.778,308.514,-69.707,-176.515,7.422,148.392
C04555=1200.782,308.265,-69.676,-176.518,7.419,148.392
C04556=1200.786,308.017,-69.647,-176.520,7.417,148.392
C04557=1200.790,307.769,-69.616,-176.523,7.413,148.392
C04558=1200.794,307.522,-69.586,-176.526,7.410,148.392
C04559=1200.799,307.273,-69.556,-176.527,7.408,148.392
C04560=1200.803,307.025,-69.525,-176.530,7.405,148.392
C04561=1200.808,306.777,-69.495,-176.533,7.402,148.392
C04562=1200.812,306.529,-69.465,-176.535,7.400,148.392
C04563=1200.816,306.280,-69.435,-176.537,7.397,148.392
C04564=1200.820,306.032,-69.405,-176.540,7.394,148.392
C04565=1200.824,305.784,-69.375,-176.542,7.391,148.392
C04566=1200.829,305.536,-69.344,-176.545,7.388,148.392
C04567=1200.833,305.288,-69.315,-176.548,7.385,148.392
C04568=1200.838,305.040,-69.284,-176.549,7.383,148.392
C04569=1200.842,304.791,-69.255,-176.552,7.380,148.392
C04570=1200.846,304.544,-69.225,-176.554,7.378,148.392
C04571=1200.851,304.295,-69.195,-176.557,7.375,148.392
C04572=1200.855,304.047,-69.165,-176.560,7.372,148.392
C04573=1200.859,303.799,-69.135,-176.562,7.370,148.392
C04574=1200.864,303.551,-69.105,-176.564,7.366,148.392
C04575=1200.867,303.303,-69.075,-176.567,7.363,148.392
C04576=1200.872,303.055,-69.045,-176.569,7.361,148.392
C04577=1200.877,302.806,-69.015,-176.572,7.358,148.392
C04578=1200.880,302.559,-68.985,-176.575,7.355,148.392
C04579=1200.884,302.310,-68.955,-176.577,7.353,148.392
C04580=1200.889,302.061,-68.925,-176.579,7.350,148.392
C04581=1200.893,301.813,-68.895,-176.582,7.348,148.392
C04582=1200.897,301.565,-68.866,-176.584,7.345,148.392
C04583=1200.901,301.317,-68.836,-176.587,7.342,148.392
C04584=1200.906,301.068,-68.806,-176.589,7.340,148.392
C04585=1200.910,300.821,-68.776,-176.592,7.337,148.392
C04586=1200.914,300.572,-68.746,-176.594,7.333,148.392
C04587=1200.918,300.324,-68.717,-176.596,7.331,148.392
C04588=1200.923,300.075,-68.687,-176.599,7.328,148.392
C04589=1200.927,299.828,-68.657,-176.602,7.325,148.392
C04590=1200.931,299.580,-68.627,-176.604,7.323,148.392
C04591=1200.936,299.332,-68.598,-176.606,7.320,148.392
C04592=1200.940,299.084,-68.569,-176.609,7.318,148.392
C04593=1200.945,298.835,-68.539,-176.611,7.315,148.392
C04594=1200.949,298.587,-68.509,-176.614,7.312,148.392
C04595=1200.953,298.339,-68.479,-176.616,7.309,148.392
C04596=1200.957,298.091,-68.450,-176.619,7.306,148.392
C04597=1200.962,297.843,-68.420,-176.621,7.304,148.392
C04598=1200.966,297.594,-68.391,-176.624,7.301,148.392
C04599=1200.971,297.346,-68.361,-176.626,7.298,148.392
C04600=1200.975,297.098,-68.331,-176.629,7.296,148.393
C04601=1200.979,296.849,-68.302,-176.632,7.293,148.393
C04602=1200.983,296.601,-68.272,-176.634,7.290,148.393
C04603=1200.987,296.353,-68.243,-176.636,7.288,148.393
C04604=1200.992,296.105,-68.213,-176.639,7.285,148.393
C04605=1200.996,295.856,-68.184,-176.641,7.283,148.393
C04606=1201.000,295.608,-68.154,-176.644,7.280,148.393
C04607=1201.005,295.360,-68.125,-176.647,7.277,148.393
C04608=1201.009,295.112,-68.096,-176.649,7.275,148.393
C04609=1201.013,294.864,-68.066,-176.651,7.272,148.393
C04610=1201.017,294.616,-68.037,-176.654,7.269,148.393
C04611=1201.022,294.367,-68.008,-176.656,7.266,148.393
C04612=1201.026,294.119,-67.978,-176.659,7.263,148.393
C04613=1201.031,293.871,-67.948,-176.661,7.261,148.393
C04614=1201.035,293.622,-67.919,-176.664,7.258,148.393
C04615=1201.040,293.375,-67.890,-176.666,7.256,148.393
C04616=1201.044,293.126,-67.860,-176.669,7.253,148.393
C04617=1201.048,292.878,-67.832,-176.671,7.250,148.393
C04618=1201.052,292.630,-67.802,-176.673,7.248,148.393
C04619=1201.056,292.381,-67.773,-176.677,7.245,148.394
C04620=1201.060,292.133,-67.744,-176.679,7.243,148.394
C04621=1201.065,291.885,-67.714,-176.681,7.240,148.394
C04622=1201.069,291.637,-67.685,-176.684,7.238,148.394
C04623=1201.074,291.388,-67.656,-176.686,7.235,148.394
C04624=1201.078,291.140,-67.627,-176.689,7.232,148.394
C04625=1201.082,290.892,-67.597,-176.691,7.229,148.394
C04626=1201.086,290.644,-67.568,-176.694,7.226,148.394
C04627=1201.091,290.395,-67.540,-176.696,7.224,148.394
C04628=1201.095,290.147,-67.510,-176.699,7.221,148.394
C04629=1201.100,289.899,-67.481,-176.702,7.219,148.394
C04630=1201.104,289.651,-67.451,-176.704,7.216,148.394
C04631=1201.108,289.403,-67.423,-176.707,7.213,148.394
C04632=1201.113,289.128,-67.390,-176.709,7.210,148.394
C04633=1201.117,288.854,-67.358,-176.712,7.207,148.394
C04634=1201.122,288.579,-67.327,-176.715,7.205,148.395
C04635=1201.127,288.305,-67.295,-176.717,7.202,148.395
C04636=1201.131,288.057,-67.266,-176.720,7.199,148.395
C04637=1201.135,287.808,-67.236,-176.723,7.196,148.395
C04638=1201.141,287.560,-67.208,-176.725,7.194,148.395
C04639=1201.145,287.312,-67.178,-176.728,7.191,148.395
C04640=1201.149,287.063,-67.150,-176.730,7.189,148.395
C04641=1201.153,286.815,-67.121,-176.733,7.186,148.395
C04642=1201.157,286.567,-67.092,-176.735,7.184,148.395
C04643=1201.162,286.319,-67.063,-176.738,7.181,148.395
C04644=1201.166,286.070,-67.034,-176.740,7.179,148.395
C04645=1201.170,285.822,-67.005,-176.743,7.176,148.395
C04646=1201.175,285.574,-66.976,-176.745,7.173,148.395
C04647=1201.179,285.325,-66.948,-176.748,7.171,148.396
C04648=1201.183,285.077,-66.918,-176.751,7.168,148.396
C04649=1201.188,284.829,-66.890,-176.753,7.166,148.396
C04650=1201.192,284.581,-66.861,-176.755,7.163,148.396
C04651=1201.196,284.332,-66.832,-176.758,7.161,148.396
C04652=1201.201,284.084,-66.804,-176.761,7.158,148.396
C04653=1201.205,283.836,-66.775,-176.763,7.156,148.396
C04654=1201.209,283.587,-66.746,-176.766,7.153,148.396
C04655=1201.214,283.339,-66.717,-176.768,7.151,148.396
C04656=1201.218,283.091,-66.689,-176.770,7.148,148.396
C04657=1201.222,282.842,-66.660,-176.773,7.145,148.396
C04658=1201.227,282.594,-66.631,-176.776,7.143,148.397
C04659=1201.231,282.346,-66.603,-176.778,7.140,148.397
C04660=1201.235,282.097,-66.574,-176.781,7.137,148.397
C04661=1201.240,281.849,-66.545,-176.783,7.134,148.397
C04662=1201.244,281.601,-66.517,-176.786,7.133,148.397
C04663=1201.249,281.353,-66.489,-176.789,7.130,148.397
C04664=1201.253,281.104,-66.461,-176.791,7.127,148.397
C04665=1201.257,280.856,-66.431,-176.793,7.124,148.397
C04666=1201.262,280.607,-66.403,-176.796,7.122,148.397
C04667=1201.266,280.359,-66.375,-176.799,7.119,148.398
C04668=1201.271,280.111,-66.346,-176.801,7.117,148.398
C04669=1201.274,279.863,-66.317,-176.804,7.114,148.398
C04670=1201.279,279.614,-66.289,-176.806,7.112,148.398
C04671=1201.283,279.366,-66.261,-176.809,7.109,148.398
C04672=1201.288,279.117,-66.232,-176.811,7.107,148.398
C04673=1201.293,278.869,-66.204,-176.814,7.104,148.398
C04674=1201.296,278.621,-66.175,-176.816,7.102,148.398
C04675=1201.301,278.372,-66.146,-176.819,7.099,148.398
C04676=1201.305,278.124,-66.118,-176.821,7.097,148.398
C04677=1201.309,277.875,-66.090,-176.824,7.094,148.398
C04678=1201.314,277.627,-66.062,-176.826,7.092,148.399
C04679=1201.318,277.379,-66.033,-176.829,7.089,148.399
C04680=1201.323,277.131,-66.005,-176.831,7.087,148.399
C04681=1201.327,276.882,-65.977,-176.834,7.084,148.399
C04682=1201.332,276.634,-65.949,-176.836,7.082,148.399
C04683=1201.335,276.385,-65.921,-176.839,7.079,148.399
C04684=1201.340,276.137,-65.892,-176.842,7.077,148.399
C04685=1201.344,275.889,-65.863,-176.844,7.074,148.399
C04686=1201.349,275.641,-65.835,-176.846,7.072,148.399
C04687=1201.353,275.392,-65.807,-176.850,7.069,148.400
C04688=1201.358,275.144,-65.779,-176.852,7.067,148.400
C04689=1201.362,274.895,-65.751,-176.854,7.064,148.400
C04690=1201.366,274.647,-65.723,-176.857,7.062,148.400
C04691=1201.371,274.398,-65.695,-176.860,7.059,148.400
C04692=1201.375,274.150,-65.667,-176.862,7.057,148.400
C04693=1201.379,273.902,-65.638,-176.865,7.054,148.400
C04694=1201.384,273.654,-65.610,-176.867,7.052,148.401
C04695=1201.388,273.405,-65.582,-176.870,7.049,148.401
C04696=1201.393,273.157,-65.554,-176.872,7.047,148.401
C04697=1201.396,272.908,-65.526,-176.875,7.045,148.401
C04698=1201.401,272.660,-65.498,-176.877,7.042,148.401
C04699=1201.405,272.412,-65.469,-176.879,7.040,148.401
C04700=1201.410,272.163,-65.442,-176.882,7.037,148.401
C04701=1201.414,271.914,-65.414,-176.885,7.035,148.401
C04702=1201.419,271.666,-65.386,-176.887,7.032,148.401
C04703=1201.423,271.418,-65.358,-176.890,7.030,148.402
C04704=1201.427,271.170,-65.330,-176.893,7.027,148.402
C04705=1201.432,270.921,-65.302,-176.895,7.025,148.402
C04706=1201.436,270.672,-65.274,-176.898,7.022,148.402
C04707=1201.440,270.425,-65.246,-176.900,7.020,148.402
C04708=1201.444,270.176,-65.218,-176.902,7.018,148.402
C04709=1201.449,269.927,-65.190,-176.905,7.015,148.402
C04710=1201.454,269.679,-65.162,-176.908,7.013,148.403
C04711=1201.458,269.431,-65.134,-176.910,7.010,148.403
C04712=1201.462,269.183,-65.107,-176.913,7.008,148.403
C04713=1201.467,268.934,-65.079,-176.916,7.005,148.403
C04714=1201.471,268.685,-65.051,-176.918,7.003,148.403
C04715=1201.475,268.438,-65.023,-176.921,7.000,148.403
C04716=1201.479,268.188,-64.996,-176.923,6.998,148.403
C04717=1201.484,267.941,-64.968,-176.925,6.996,148.403
C04718=1201.489,267.692,-64.940,-176.928,6.993,148.404
C04719=1201.493,267.443,-64.912,-176.931,6.991,148.404
C04720=1201.497,267.195,-64.884,-176.933,6.988,148.404
C04721=1201.502,266.947,-64.857,-176.936,6.986,148.404
C04722=1201.506,266.698,-64.829,-176.939,6.983,148.404
C04723=1201.510,266.450,-64.802,-176.941,6.981,148.404
C04724=1201.515,266.202,-64.774,-176.943,6.979,148.405
C04725=1201.520,265.952,-64.746,-176.946,6.976,148.405
C04726=1201.524,265.704,-64.718,-176.948,6.974,148.405
C04727=1201.529,265.456,-64.691,-176.952,6.971,148.405
C04728=1201.532,265.207,-64.663,-176.954,6.969,148.405
C04729=1201.537,264.959,-64.636,-176.956,6.966,148.405
C04730=1201.541,264.711,-64.608,-176.959,6.964,148.405
C04731=1201.546,264.463,-64.581,-176.961,6.962,148.405
C04732=1201.550,264.214,-64.553,-176.964,6.959,148.406
C04733=1201.554,263.965,-64.526,-176.966,6.957,148.406
C04734=1201.559,263.718,-64.498,-176.969,6.954,148.406
C04735=1201.563,263.468,-64.470,-176.972,6.952,148.406
C04736=1201.568,263.196,-64.441,-176.974,6.949,148.406
C04737=1201.573,262.923,-64.410,-176.977,6.947,148.407
C04738=1201.577,262.650,-64.380,-176.980,6.944,148.407
C04739=1201.582,262.377,-64.350,-176.983,6.942,148.407
C04740=1201.587,262.129,-64.323,-176.985,6.939,148.407
C04741=1201.592,261.880,-64.296,-176.988,6.937,148.407
C04742=1201.596,261.632,-64.268,-176.990,6.935,148.407
C04743=1201.600,261.383,-64.241,-176.993,6.933,148.408
C04744=1201.605,261.135,-64.213,-176.996,6.930,148.408
C04745=1201.609,260.887,-64.186,-176.998,6.928,148.408
C04746=1201.613,260.638,-64.158,-177.001,6.925,148.408
C04747=1201.618,260.389,-64.131,-177.003,6.923,148.408
C04748=1201.622,260.141,-64.103,-177.006,6.921,148.408
C04749=1201.627,259.893,-64.076,-177.009,6.918,148.408
C04750=1201.632,259.644,-64.049,-177.011,6.916,148.408
C04751=1201.636,259.395,-64.022,-177.013,6.914,148.409
C04752=1201.640,259.147,-63.995,-177.016,6.911,148.409
C04753=1201.644,258.899,-63.968,-177.019,6.909,148.409
C04754=1201.649,258.651,-63.941,-177.021,6.906,148.409
C04755=1201.653,258.402,-63.913,-177.024,6.904,148.409
C04756=1201.658,258.154,-63.886,-177.026,6.902,148.410
C04757=1201.662,257.905,-63.859,-177.029,6.899,148.410
C04758=1201.667,257.656,-63.832,-177.032,6.897,148.410
C04759=1201.671,257.408,-63.804,-177.034,6.895,148.410
C04760=1201.676,257.160,-63.777,-177.037,6.892,148.410
C04761=1201.680,256.911,-63.751,-177.039,6.890,148.410
C04762=1201.684,256.663,-63.724,-177.042,6.888,148.411
C04763=1201.688,256.414,-63.696,-177.044,6.885,148.411
C04764=1201.693,256.165,-63.669,-177.047,6.883,148.411
C04765=1201.698,255.917,-63.642,-177.050,6.880,148.411
C04766=1201.701,255.669,-63.616,-177.052,6.878,148.411
C04767=1201.706,255.420,-63.589,-177.054,6.876,148.411
C04768=1201.711,255.172,-63.561,-177.058,6.874,148.412
C04769=1201.715,254.923,-63.534,-177.060,6.871,148.412
C04770=1201.720,254.675,-63.507,-177.062,6.870,148.412
C04771=1201.723,254.426,-63.480,-177.065,6.867,148.412
C04772=1201.728,254.177,-63.453,-177.067,6.864,148.412
C04773=1201.733,253.929,-63.426,-177.070,6.863,148.413
C04774=1201.737,253.680,-63.399,-177.073,6.860,148.413
C04775=1201.741,253.432,-63.373,-177.075,6.858,148.413
C04776=1201.746,253.184,-63.346,-177.077,6.856,148.413
C04777=1201.751,252.935,-63.319,-177.081,6.853,148.413
C04778=1201.755,252.687,-63.292,-177.083,6.851,148.413
C04779=1201.759,252.438,-63.265,-177.085,6.849,148.414
C04780=1201.764,252.190,-63.238,-177.088,6.846,148.414
C04781=1201.769,251.941,-63.212,-177.091,6.844,148.414
C04782=1201.773,251.693,-63.185,-177.093,6.842,148.414
C04783=1201.777,251.444,-63.158,-177.096,6.839,148.414
C04784=1201.782,251.196,-63.131,-177.098,6.837,148.415
C04785=1201.785,250.947,-63.104,-177.101,6.835,148.415
C04786=1201.790,250.698,-63.077,-177.103,6.833,148.415
C04787=1201.795,250.449,-63.051,-177.106,6.830,148.415
C04788=1201.799,250.201,-63.024,-177.108,6.828,148.415
C04789=1201.804,249.952,-62.997,-177.111,6.826,148.416
C04790=1201.807,249.704,-62.971,-177.114,6.823,148.416
C04791=1201.812,249.455,-62.945,-177.116,6.821,148.416
C04792=1201.817,249.207,-62.918,-177.119,6.820,148.416
C04793=1201.821,248.958,-62.891,-177.122,6.817,148.416
C04794=1201.826,248.710,-62.864,-177.124,6.815,148.417
C04795=1201.830,248.461,-62.838,-177.126,6.812,148.417
C04796=1201.835,248.213,-62.811,-177.129,6.811,148.417
C04797=1201.839,247.964,-62.784,-177.132,6.808,148.417
C04798=1201.843,247.715,-62.758,-177.134,6.806,148.417
C04799=1201.848,247.467,-62.731,-177.136,6.804,148.418
C04800=1201.852,247.219,-62.705,-177.140,6.801,148.418
C04801=1201.858,246.970,-62.679,-177.142,6.799,148.418
C04802=1201.861,246.722,-62.652,-177.144,6.797,148.418
C04803=1201.866,246.474,-62.625,-177.147,6.794,148.418
C04804=1201.870,246.225,-62.600,-177.150,6.792,148.419
C04805=1201.875,245.976,-62.573,-177.152,6.790,148.419
C04806=1201.879,245.727,-62.547,-177.155,6.788,148.419
C04807=1201.884,245.479,-62.520,-177.158,6.785,148.419
C04808=1201.888,245.230,-62.494,-177.160,6.783,148.419
C04809=1201.893,244.982,-62.467,-177.163,6.781,148.420
C04810=1201.897,244.733,-62.441,-177.165,6.779,148.420
C04811=1201.902,244.484,-62.414,-177.168,6.777,148.420
C04812=1201.906,244.236,-62.388,-177.170,6.774,148.420
C04813=1201.911,243.987,-62.361,-177.173,6.773,148.420
C04814=1201.915,243.738,-62.336,-177.176,6.770,148.421
C04815=1201.919,243.491,-62.309,-177.178,6.768,148.421
C04816=1201.924,243.242,-62.283,-177.181,6.766,148.421
C04817=1201.928,242.994,-62.257,-177.183,6.764,148.421
C04818=1201.933,242.744,-62.230,-177.186,6.761,148.422
C04819=1201.937,242.496,-62.204,-177.188,6.759,148.422
C04820=1201.941,242.247,-62.178,-177.191,6.757,148.422
C04821=1201.946,241.998,-62.152,-177.193,6.755,148.422
C04822=1201.950,241.750,-62.125,-177.196,6.752,148.422
C04823=1201.956,241.502,-62.099,-177.199,6.750,148.423
C04824=1201.960,241.254,-62.073,-177.201,6.748,148.423
C04825=1201.964,241.005,-62.047,-177.204,6.746,148.423
C04826=1201.969,240.756,-62.021,-177.207,6.744,148.423
C04827=1201.973,240.507,-61.994,-177.209,6.741,148.423
C04828=1201.977,240.259,-61.969,-177.212,6.740,148.424
C04829=1201.982,240.009,-61.942,-177.214,6.737,148.424
C04830=1201.986,239.762,-61.916,-177.217,6.735,148.424
C04831=1201.991,239.513,-61.890,-177.219,6.733,148.424
C04832=1201.995,239.264,-61.865,-177.222,6.731,148.425
C04833=1202.000,239.015,-61.838,-177.224,6.729,148.425
C04834=1202.004,238.767,-61.812,-177.226,6.727,148.425
C04835=1202.009,238.519,-61.786,-177.230,6.724,148.425
C04836=1202.014,238.270,-61.760,-177.232,6.722,148.426
C04837=1202.018,238.021,-61.734,-177.234,6.720,148.426
C04838=1202.022,237.772,-61.709,-177.237,6.718,148.426
C04839=1202.026,237.524,-61.682,-177.240,6.716,148.426
C04840=1202.032,237.253,-61.654,-177.242,6.713,148.426
C04841=1202.036,236.981,-61.625,-177.246,6.711,148.427
C04842=1202.041,236.709,-61.597,-177.248,6.709,148.427
C04843=1202.046,236.438,-61.569,-177.251,6.706,148.427
C04844=1202.051,236.189,-61.544,-177.254,6.704,148.427
C04845=1202.054,235.941,-61.517,-177.256,6.702,148.428
C04846=1202.059,235.692,-61.491,-177.259,6.700,148.428
C04847=1202.064,235.444,-61.465,-177.262,6.697,148.428
C04848=1202.068,235.195,-61.440,-177.264,6.695,148.428
C04849=1202.073,234.946,-61.414,-177.267,6.694,148.429
C04850=1202.078,234.698,-61.388,-177.269,6.691,148.429
C04851=1202.082,234.449,-61.363,-177.272,6.690,148.429
C04852=1202.086,234.201,-61.337,-177.275,6.687,148.429
C04853=1202.091,233.952,-61.311,-177.277,6.685,148.430
C04854=1202.096,233.703,-61.285,-177.280,6.683,148.430
C04855=1202.100,233.455,-61.259,-177.282,6.681,148.430
C04856=1202.104,233.206,-61.234,-177.284,6.679,148.430
C04857=1202.109,232.958,-61.208,-177.288,6.676,148.431
C04858=1202.113,232.709,-61.183,-177.290,6.674,148.431
C04859=1202.118,232.460,-61.157,-177.292,6.672,148.431
C04860=1202.122,232.211,-61.131,-177.295,6.670,148.431
C04861=1202.127,231.963,-61.106,-177.298,6.669,148.432
C04862=1202.131,231.714,-61.080,-177.300,6.666,148.432
C04863=1202.136,231.465,-61.054,-177.303,6.664,148.432
C04864=1202.141,231.217,-61.028,-177.306,6.662,148.432
C04865=1202.145,230.968,-61.003,-177.308,6.660,148.432
C04866=1202.149,230.719,-60.977,-177.310,6.658,148.433
C04867=1202.154,230.471,-60.952,-177.313,6.656,148.433
C04868=1202.158,230.222,-60.926,-177.316,6.653,148.433
C04869=1202.163,229.974,-60.901,-177.318,6.651,148.433
C04870=1202.167,229.725,-60.875,-177.321,6.649,148.434
C04871=1202.172,229.476,-60.849,-177.323,6.647,148.434
C04872=1202.177,229.228,-60.825,-177.326,6.645,148.434
C04873=1202.181,228.979,-60.799,-177.329,6.644,148.435
C04874=1202.185,228.730,-60.773,-177.332,6.641,148.435
C04875=1202.190,228.482,-60.748,-177.334,6.639,148.435
C04876=1202.195,228.232,-60.723,-177.337,6.637,148.435
C04877=1202.199,227.984,-60.697,-177.339,6.635,148.436
C04878=1202.203,227.736,-60.672,-177.341,6.633,148.436
C04879=1202.207,227.487,-60.647,-177.345,6.630,148.436
C04880=1202.212,227.238,-60.622,-177.347,6.628,148.436
C04881=1202.216,226.990,-60.596,-177.350,6.627,148.437
C04882=1202.221,226.741,-60.571,-177.352,6.624,148.437
C04883=1202.226,226.492,-60.546,-177.355,6.623,148.437
C04884=1202.230,226.243,-60.520,-177.357,6.621,148.437
C04885=1202.235,225.995,-60.495,-177.359,6.619,148.438
C04886=1202.239,225.746,-60.470,-177.363,6.616,148.438
C04887=1202.244,225.498,-60.444,-177.365,6.614,148.438
C04888=1202.248,225.249,-60.419,-177.368,6.612,148.438
C04889=1202.253,225.000,-60.394,-177.370,6.610,148.439
C04890=1202.257,224.752,-60.369,-177.373,6.608,148.439
C04891=1202.262,224.503,-60.343,-177.375,6.606,148.439
C04892=1202.266,224.254,-60.318,-177.378,6.604,148.440
C04893=1202.271,224.006,-60.293,-177.381,6.602,148.440
C04894=1202.276,223.756,-60.268,-177.383,6.600,148.440
C04895=1202.280,223.509,-60.243,-177.386,6.598,148.440
C04896=1202.284,223.259,-60.218,-177.389,6.596,148.441
C04897=1202.289,223.010,-60.192,-177.391,6.594,148.441
C04898=1202.294,222.762,-60.167,-177.393,6.592,148.441
C04899=1202.298,222.513,-60.142,-177.397,6.589,148.441
C04900=1202.302,222.265,-60.118,-177.399,6.588,148.442
C04901=1202.307,222.016,-60.092,-177.401,6.585,148.442
C04902=1202.312,221.767,-60.067,-177.404,6.584,148.442
C04903=1202.317,221.519,-60.042,-177.407,6.582,148.442
C04904=1202.320,221.270,-60.017,-177.409,6.580,148.443
C04905=1202.325,221.022,-59.992,-177.412,6.578,148.443
C04906=1202.330,220.772,-59.967,-177.414,6.576,148.443
C04907=1202.334,220.524,-59.943,-177.417,6.573,148.443
C04908=1202.338,220.275,-59.917,-177.420,6.571,148.444
C04909=1202.343,220.026,-59.892,-177.423,6.570,148.444
C04910=1202.348,219.778,-59.867,-177.425,6.567,148.444
C04911=1202.352,219.529,-59.843,-177.427,6.566,148.445
C04912=1202.357,219.280,-59.818,-177.430,6.564,148.445
C04913=1202.361,219.032,-59.792,-177.433,6.562,148.445
C04914=1202.365,218.782,-59.768,-177.435,6.560,148.446
C04915=1202.370,218.534,-59.743,-177.438,6.557,148.446
C04916=1202.375,218.286,-59.718,-177.441,6.555,148.446
C04917=1202.379,218.037,-59.693,-177.443,6.553,148.446
C04918=1202.384,217.788,-59.669,-177.446,6.552,148.447
C04919=1202.389,217.538,-59.644,-177.449,6.550,148.447
C04920=1202.393,217.291,-59.619,-177.451,6.548,148.447
C04921=1202.398,217.042,-59.594,-177.453,6.546,148.447
C04922=1202.402,216.793,-59.570,-177.456,6.544,148.448
C04923=1202.407,216.544,-59.545,-177.459,6.541,148.448
C04924=1202.411,216.295,-59.519,-177.462,6.539,148.448
C04925=1202.415,216.047,-59.495,-177.464,6.537,148.449
C04926=1202.421,215.798,-59.471,-177.467,6.535,148.449
C04927=1202.424,215.549,-59.446,-177.469,6.534,148.449
C04928=1202.429,215.300,-59.421,-177.472,6.532,148.450
C04929=1202.434,215.052,-59.397,-177.475,6.530,148.450
C04930=1202.438,214.803,-59.372,-177.477,6.528,148.450
C04931=1202.442,214.555,-59.348,-177.479,6.526,148.450
C04932=1202.447,214.305,-59.323,-177.482,6.524,148.451
C04933=1202.452,214.056,-59.298,-177.485,6.522,148.451
C04934=1202.457,213.808,-59.274,-177.488,6.520,148.451
C04935=1202.461,213.559,-59.249,-177.491,6.518,148.452
C04936=1202.465,213.310,-59.225,-177.493,6.516,148.452
C04937=1202.471,213.061,-59.200,-177.495,6.514,148.452
C04938=1202.474,212.812,-59.176,-177.498,6.512,148.452
C04939=1202.479,212.564,-59.150,-177.501,6.510,148.453
C04940=1202.484,212.316,-59.126,-177.503,6.508,148.453
C04941=1202.489,212.067,-59.101,-177.506,6.507,148.453
C04942=1202.493,211.818,-59.077,-177.509,6.505,148.454
C04943=1202.497,211.570,-59.053,-177.511,6.503,148.454
C04944=1202.502,211.299,-59.027,-177.515,6.500,148.454
C04945=1202.507,211.028,-59.000,-177.517,6.498,148.455
C04946=1202.512,210.758,-58.973,-177.520,6.497,148.455
C04947=1202.517,210.488,-58.946,-177.523,6.494,148.455
C04948=1202.522,210.239,-58.922,-177.525,6.492,148.455
C04949=1202.526,209.990,-58.897,-177.528,6.490,148.456
C04950=1202.531,209.741,-58.873,-177.530,6.488,148.456
C04951=1202.535,209.492,-58.850,-177.533,6.486,148.456
C04952=1202.540,209.244,-58.825,-177.536,6.484,148.457
C04953=1202.544,208.994,-58.801,-177.538,6.483,148.457
C04954=1202.549,208.746,-58.777,-177.541,6.481,148.458
C04955=1202.554,208.497,-58.752,-177.543,6.479,148.458
C04956=1202.558,208.249,-58.728,-177.546,6.477,148.458
C04957=1202.563,208.000,-58.703,-177.549,6.475,148.458
C04958=1202.567,207.750,-58.680,-177.552,6.472,148.459
C04959=1202.572,207.502,-58.655,-177.554,6.471,148.459
C04960=1202.577,207.253,-58.631,-177.557,6.469,148.459
C04961=1202.581,207.005,-58.607,-177.560,6.467,148.460
C04962=1202.585,206.756,-58.582,-177.562,6.465,148.460
C04963=1202.590,206.507,-58.559,-177.565,6.463,148.460
C04964=1202.595,206.258,-58.534,-177.567,6.461,148.460
C04965=1202.599,206.010,-58.510,-177.570,6.459,148.461
C04966=1202.604,205.761,-58.486,-177.572,6.457,148.461
C04967=1202.609,205.512,-58.462,-177.575,6.456,148.461
C04968=1202.613,205.263,-58.438,-177.578,6.454,148.462
C04969=1202.617,205.014,-58.414,-177.580,6.452,148.462
C04970=1202.622,204.766,-58.390,-177.583,6.450,148.462
C04971=1202.627,204.517,-58.366,-177.586,6.448,148.463
C04972=1202.632,204.268,-58.342,-177.588,6.446,148.463
C04973=1202.635,204.019,-58.317,-177.590,6.444,148.463
C04974=1202.640,203.770,-58.294,-177.593,6.443,148.464
C04975=1202.644,203.522,-58.270,-177.596,6.441,148.464
C04976=1202.650,203.272,-58.246,-177.598,6.439,148.464
C04977=1202.654,203.024,-58.222,-177.601,6.437,148.465
C04978=1202.659,202.775,-58.198,-177.604,6.435,148.465
C04979=1202.663,202.526,-58.174,-177.606,6.433,148.465
C04980=1202.667,202.277,-58.150,-177.609,6.432,148.466
C04981=1202.673,202.028,-58.126,-177.612,6.430,148.466
C04982=1202.677,201.780,-58.102,-177.614,6.428,148.466
C04983=1202.681,201.531,-58.078,-177.617,6.426,148.467
C04984=1202.686,201.282,-58.054,-177.619,6.424,148.467
C04985=1202.690,201.034,-58.030,-177.622,6.422,148.467
C04986=1202.695,200.785,-58.007,-177.624,6.420,148.467
C04987=1202.700,200.536,-57.983,-177.627,6.419,148.468
C04988=1202.704,200.287,-57.959,-177.630,6.417,148.468
C04989=1202.709,200.039,-57.935,-177.632,6.415,148.469
C04990=1202.713,199.789,-57.911,-177.635,6.413,148.469
C04991=1202.718,199.540,-57.887,-177.638,6.411,148.469
C04992=1202.723,199.291,-57.864,-177.640,6.409,148.470
C04993=1202.727,199.042,-57.840,-177.643,6.408,148.470
C04994=1202.732,198.794,-57.816,-177.646,6.406,148.470
C04995=1202.736,198.545,-57.793,-177.648,6.404,148.471
C04996=1202.741,198.296,-57.769,-177.651,6.402,148.471
C04997=1202.745,198.047,-57.745,-177.654,6.400,148.471
C04998=1202.750,197.798,-57.722,-177.656,6.398,148.472
C04999=1202.755,197.550,-57.698,-177.658,6.396,148.472
C05000=1202.759,197.301,-57.675,-177.661,6.395,148.472
C05001=1202.764,197.053,-57.651,-177.664,6.393,148.472
C05002=1202.768,196.803,-57.627,-177.666,6.391,148.473
C05003=1202.773,196.554,-57.604,-177.669,6.389,148.473
C05004=1202.777,196.306,-57.580,-177.672,6.387,148.473
C05005=1202.782,196.057,-57.556,-177.674,6.385,148.474
C05006=1202.787,195.808,-57.533,-177.677,6.384,148.474
C05007=1202.792,195.559,-57.510,-177.680,6.382,148.475
C05008=1202.796,195.311,-57.486,-177.682,6.380,148.475
C05009=1202.801,195.062,-57.462,-177.685,6.378,148.475
C05010=1202.805,194.812,-57.439,-177.688,6.376,148.476
C05011=1202.810,194.563,-57.415,-177.690,6.375,148.476
C05012=1202.814,194.315,-57.391,-177.693,6.373,148.476
C05013=1202.819,194.066,-57.368,-177.696,6.371,148.477
C05014=1202.824,193.817,-57.345,-177.698,6.369,148.477
C05015=1202.829,193.568,-57.321,-177.701,6.367,148.477
C05016=1202.833,193.320,-57.297,-177.704,6.365,148.478
C05017=1202.838,193.070,-57.274,-177.706,6.364,148.478
C05018=1202.842,192.821,-57.251,-177.709,6.362,148.478
C05019=1202.846,192.573,-57.228,-177.712,6.360,148.479
C05020=1202.851,192.324,-57.204,-177.714,6.358,148.479
C05021=1202.856,192.075,-57.181,-177.717,6.356,148.479
C05022=1202.860,191.826,-57.158,-177.719,6.355,148.480
C05023=1202.865,191.578,-57.134,-177.722,6.354,148.480
C05024=1202.870,191.329,-57.111,-177.724,6.352,148.480
C05025=1202.875,191.080,-57.087,-177.727,6.350,148.481
C05026=1202.879,190.831,-57.065,-177.730,6.348,148.481
C05027=1202.883,190.582,-57.041,-177.732,6.346,148.482
C05028=1202.888,190.333,-57.018,-177.735,6.344,148.482
C05029=1202.893,190.084,-56.994,-177.738,6.343,148.482
C05030=1202.898,189.835,-56.971,-177.740,6.341,148.483
C05031=1202.902,189.586,-56.948,-177.743,6.339,148.483
C05032=1202.906,189.337,-56.925,-177.746,6.337,148.483
C05033=1202.912,189.089,-56.902,-177.748,6.335,148.484
C05034=1202.916,188.840,-56.879,-177.751,6.334,148.484
C05035=1202.921,188.591,-56.855,-177.753,6.332,148.484
C05036=1202.925,188.342,-56.832,-177.756,6.330,148.485
C05037=1202.930,188.093,-56.809,-177.758,6.329,148.485
C05038=1202.934,187.844,-56.786,-177.761,6.327,148.485
C05039=1202.939,187.595,-56.762,-177.764,6.325,148.486
C05040=1202.944,187.347,-56.740,-177.766,6.324,148.486
C05041=1202.948,187.098,-56.717,-177.769,6.322,148.486
C05042=1202.953,186.849,-56.693,-177.772,6.320,148.487
C05043=1202.958,186.599,-56.671,-177.774,6.318,148.487
C05044=1202.962,186.351,-56.648,-177.777,6.316,148.488
C05045=1202.967,186.102,-56.625,-177.780,6.314,148.488
C05046=1202.971,185.853,-56.601,-177.782,6.313,148.488
C05047=1202.976,185.605,-56.579,-177.785,6.311,148.489
C05048=1202.981,185.335,-56.554,-177.787,6.309,148.489
C05049=1202.987,185.065,-56.529,-177.790,6.307,148.489
C05050=1202.991,184.796,-56.504,-177.793,6.305,148.490
C05051=1202.996,184.526,-56.479,-177.796,6.304,148.490
C05052=1203.000,184.277,-56.456,-177.799,6.302,148.491
C05053=1203.005,184.028,-56.433,-177.801,6.300,148.491
C05054=1203.010,183.779,-56.410,-177.804,6.299,148.491
C05055=1203.014,183.530,-56.388,-177.807,6.297,148.492
C05056=1203.019,183.281,-56.365,-177.809,6.295,148.492
C05057=1203.023,183.033,-56.342,-177.812,6.293,148.492
C05058=1203.028,182.784,-56.319,-177.814,6.292,148.493
C05059=1203.033,182.534,-56.296,-177.817,6.290,148.493
C05060=1203.038,182.286,-56.274,-177.819,6.288,148.493
C05061=1203.042,182.037,-56.250,-177.822,6.287,148.494
C05062=1203.047,181.787,-56.228,-177.825,6.285,148.494
C05063=1203.051,181.538,-56.205,-177.827,6.283,148.495
C05064=1203.057,181.290,-56.182,-177.830,6.281,148.495
C05065=1203.061,181.041,-56.160,-177.833,6.279,148.495
C05066=1203.065,180.792,-56.136,-177.835,6.278,148.496
C05067=1203.069,180.543,-56.114,-177.837,6.277,148.496
C05068=1203.075,180.294,-56.091,-177.840,6.275,148.496
C05069=1203.079,180.045,-56.069,-177.843,6.273,148.497
C05070=1203.084,179.796,-56.046,-177.846,6.272,148.497
C05071=1203.089,179.548,-56.024,-177.849,6.270,148.498
C05072=1203.093,179.299,-56.000,-177.851,6.268,148.498
C05073=1203.098,179.049,-55.978,-177.854,6.266,148.498
C05074=1203.102,178.800,-55.955,-177.856,6.265,148.499
C05075=1203.107,178.552,-55.933,-177.859,6.263,148.499
C05076=1203.112,178.303,-55.910,-177.861,6.262,148.499
C05077=1203.116,178.053,-55.888,-177.864,6.260,148.500
C05078=1203.121,177.805,-55.865,-177.867,6.258,148.500
C05079=1203.126,177.556,-55.843,-177.869,6.256,148.501
C05080=1203.130,177.307,-55.820,-177.871,6.255,148.501
C05081=1203.135,177.058,-55.798,-177.874,6.253,148.501
C05082=1203.139,176.809,-55.775,-177.877,6.252,148.502
C05083=1203.144,176.560,-55.752,-177.880,6.250,148.502
C05084=1203.149,176.312,-55.730,-177.882,6.248,148.503
C05085=1203.153,176.062,-55.708,-177.885,6.246,148.503
C05086=1203.158,175.813,-55.684,-177.888,6.245,148.503
C05087=1203.163,175.565,-55.663,-177.890,6.244,148.504
C05088=1203.168,175.315,-55.640,-177.893,6.242,148.504
C05089=1203.172,175.067,-55.618,-177.895,6.240,148.504
C05090=1203.176,174.818,-55.596,-177.898,6.238,148.505
C05091=1203.181,174.568,-55.572,-177.901,6.236,148.505
C05092=1203.186,174.320,-55.551,-177.903,6.235,148.505
C05093=1203.190,174.070,-55.529,-177.905,6.234,148.506
C05094=1203.196,173.822,-55.506,-177.908,6.232,148.506
C05095=1203.200,173.573,-55.483,-177.911,6.230,148.507
C05096=1203.204,173.323,-55.461,-177.914,6.229,148.507
C05097=1203.209,173.075,-55.438,-177.916,6.227,148.508
C05098=1203.214,172.826,-55.416,-177.919,6.226,148.508
C05099=1203.219,172.577,-55.395,-177.921,6.224,148.508
C05100=1203.223,172.328,-55.371,-177.924,6.222,148.509
C05101=1203.228,172.079,-55.349,-177.927,6.220,148.509
C05102=1203.232,171.830,-55.328,-177.929,6.219,148.509
C05103=1203.237,171.580,-55.305,-177.932,6.217,148.510
C05104=1203.242,171.332,-55.283,-177.934,6.216,148.510
C05105=1203.246,171.083,-55.261,-177.937,6.214,148.511
C05106=1203.251,170.835,-55.239,-177.940,6.213,148.511
C05107=1203.256,170.585,-55.216,-177.942,6.211,148.511
C05108=1203.261,170.336,-55.195,-177.945,6.209,148.512
C05109=1203.265,170.087,-55.172,-177.947,6.208,148.512
C05110=1203.270,169.839,-55.150,-177.950,6.206,148.513
C05111=1203.275,169.589,-55.127,-177.953,6.205,148.513
C05112=1203.280,169.341,-55.106,-177.956,6.203,148.513
C05113=1203.284,169.091,-55.084,-177.958,6.201,148.514
C05114=1203.288,168.842,-55.062,-177.961,6.200,148.514
C05115=1203.293,168.593,-55.040,-177.963,6.198,148.515
C05116=1203.298,168.344,-55.017,-177.966,6.197,148.515
C05117=1203.303,168.096,-54.995,-177.969,6.195,148.515
C05118=1203.307,167.846,-54.973,-177.972,6.193,148.516
C05119=1203.312,167.598,-54.951,-177.974,6.192,148.516
C05120=1203.317,167.349,-54.929,-177.976,6.190,148.517
C05121=1203.321,167.100,-54.907,-177.979,6.189,148.517
C05122=1203.327,166.851,-54.885,-177.982,6.187,148.517
C05123=1203.331,166.601,-54.863,-177.984,6.186,148.518
C05124=1203.336,166.353,-54.841,-177.987,6.184,148.518
C05125=1203.340,166.103,-54.819,-177.990,6.183,148.519
C05126=1203.345,165.855,-54.798,-177.992,6.181,148.519
C05127=1203.349,165.605,-54.776,-177.995,6.179,148.519
C05128=1203.354,165.357,-54.754,-177.997,6.178,148.520
C05129=1203.358,165.107,-54.732,-178.000,6.176,148.520
C05130=1203.363,164.859,-54.710,-178.002,6.174,148.521
C05131=1203.367,164.609,-54.688,-178.006,6.173,148.521
C05132=1203.372,164.361,-54.667,-178.008,6.172,148.522
C05133=1203.378,164.112,-54.644,-178.010,6.170,148.522
C05134=1203.382,163.862,-54.622,-178.013,6.168,148.522
C05135=1203.387,163.614,-54.601,-178.016,6.167,148.523
C05136=1203.391,163.364,-54.578,-178.018,6.166,148.523
C05137=1203.396,163.115,-54.557,-178.021,6.164,148.524
C05138=1203.401,162.866,-54.535,-178.024,6.162,148.524
C05139=1203.406,162.617,-54.514,-178.026,6.161,148.524
C05140=1203.410,162.369,-54.492,-178.028,6.160,148.525
C05141=1203.415,162.119,-54.470,-178.031,6.158,148.525
C05142=1203.420,161.871,-54.448,-178.034,6.156,148.526
C05143=1203.424,161.621,-54.426,-178.037,6.155,148.526
C05144=1203.429,161.372,-54.405,-178.039,6.154,148.527
C05145=1203.434,161.123,-54.384,-178.042,6.152,148.527
C05146=1203.438,160.874,-54.362,-178.044,6.150,148.527
C05147=1203.443,160.625,-54.340,-178.047,6.148,148.528
C05148=1203.448,160.377,-54.318,-178.050,6.148,148.528
C05149=1203.452,160.127,-54.297,-178.052,6.146,148.529
C05150=1203.457,159.878,-54.276,-178.055,6.144,148.529
C05151=1203.461,159.630,-54.254,-178.058,6.142,148.529
C05152=1203.467,159.360,-54.231,-178.061,6.141,148.530
C05153=1203.472,159.091,-54.207,-178.063,6.140,148.530
C05154=1203.477,158.823,-54.184,-178.066,6.138,148.531
C05155=1203.482,158.553,-54.161,-178.069,6.137,148.531
C05156=1203.486,158.304,-54.139,-178.071,6.135,148.532
C05157=1203.491,158.055,-54.118,-178.074,6.133,148.532
C05158=1203.496,157.806,-54.096,-178.077,6.131,148.532
C05159=1203.500,157.557,-54.074,-178.079,6.131,148.533
C05160=1203.505,157.308,-54.053,-178.082,6.129,148.533
C05161=1203.510,157.059,-54.032,-178.085,6.127,148.534
C05162=1203.514,156.810,-54.010,-178.087,6.126,148.534
C05163=1203.520,156.561,-53.989,-178.089,6.124,148.535
C05164=1203.524,156.312,-53.968,-178.093,6.123,148.535
C05165=1203.529,156.063,-53.947,-178.095,6.121,148.536
C05166=1203.533,155.814,-53.925,-178.097,6.120,148.536
C05167=1203.538,155.565,-53.903,-178.100,6.118,148.536
C05168=1203.543,155.316,-53.882,-178.103,6.116,148.537
C05169=1203.548,155.067,-53.860,-178.105,6.116,148.537
C05170=1203.552,154.817,-53.840,-178.108,6.114,148.538
C05171=1203.557,154.569,-53.818,-178.111,6.112,148.538
C05172=1203.562,154.320,-53.797,-178.113,6.111,148.538
C05173=1203.566,154.070,-53.775,-178.116,6.110,148.539
C05174=1203.571,153.821,-53.755,-178.119,6.108,148.539
C05175=1203.576,153.573,-53.733,-178.121,6.106,148.540
C05176=1203.581,153.323,-53.712,-178.123,6.105,148.540
C05177=1203.586,153.075,-53.690,-178.127,6.104,148.541
C05178=1203.590,152.825,-53.669,-178.129,6.102,148.541
C05179=1203.594,152.576,-53.648,-178.131,6.101,148.542
C05180=1203.600,152.327,-53.627,-178.134,6.099,148.542
C05181=1203.604,152.078,-53.605,-178.137,6.097,148.542
C05182=1203.608,151.829,-53.584,-178.139,6.097,148.543
C05183=1203.613,151.580,-53.563,-178.142,6.095,148.543
C05184=1203.618,151.331,-53.542,-178.145,6.093,148.544
C05185=1203.623,151.082,-53.521,-178.147,6.092,148.544
C05186=1203.628,150.833,-53.500,-178.150,6.091,148.545
C05187=1203.633,150.584,-53.479,-178.153,6.089,148.545
C05188=1203.637,150.334,-53.457,-178.155,6.088,148.545
C05189=1203.641,150.086,-53.436,-178.157,6.086,148.546
C05190=1203.647,149.837,-53.415,-178.161,6.085,148.546
C05191=1203.652,149.587,-53.394,-178.163,6.084,148.547
C05192=1203.656,149.339,-53.373,-178.165,6.082,148.547
C05193=1203.661,149.089,-53.352,-178.169,6.081,148.548
C05194=1203.666,148.840,-53.331,-178.171,6.080,148.548
C05195=1203.670,148.591,-53.310,-178.173,6.078,148.549
C05196=1203.675,148.342,-53.289,-178.176,6.076,148.549
C05197=1203.679,148.093,-53.269,-178.179,6.076,148.550
C05198=1203.685,147.844,-53.248,-178.181,6.074,148.550
C05199=1203.689,147.595,-53.226,-178.184,6.072,148.550
C05200=1203.693,147.346,-53.205,-178.186,6.071,148.551
C05201=1203.698,147.096,-53.184,-178.189,6.070,148.551
C05202=1203.703,146.847,-53.164,-178.192,6.068,148.552
C05203=1203.708,146.599,-53.142,-178.194,6.067,148.552
C05204=1203.713,146.350,-53.121,-178.197,6.065,148.553
C05205=1203.717,146.101,-53.101,-178.200,6.064,148.553
C05206=1203.723,145.851,-53.080,-178.202,6.063,148.553
C05207=1203.727,145.602,-53.059,-178.205,6.061,148.554
C05208=1203.732,145.353,-53.038,-178.207,6.060,148.554
C05209=1203.736,145.104,-53.017,-178.210,6.058,148.555
C05210=1203.741,144.855,-52.996,-178.213,6.057,148.555
C05211=1203.745,144.606,-52.976,-178.215,6.056,148.556
C05212=1203.751,144.357,-52.955,-178.218,6.054,148.556
C05213=1203.755,144.108,-52.934,-178.221,6.052,148.557
C05214=1203.760,143.858,-52.913,-178.223,6.051,148.557
C05215=1203.765,143.609,-52.893,-178.226,6.050,148.558
C05216=1203.770,143.360,-52.872,-178.229,6.048,148.558
C05217=1203.774,143.111,-52.852,-178.231,6.047,148.558
C05218=1203.779,142.863,-52.830,-178.234,6.046,148.559
C05219=1203.783,142.614,-52.810,-178.236,6.045,148.559
C05220=1203.789,142.364,-52.789,-178.239,6.043,148.560
C05221=1203.793,142.115,-52.768,-178.241,6.041,148.560
C05222=1203.798,141.867,-52.748,-178.244,6.041,148.561
C05223=1203.803,141.617,-52.727,-178.247,6.039,148.561
C05224=1203.807,141.368,-52.707,-178.249,6.038,148.562
C05225=1203.812,141.119,-52.686,-178.252,6.037,148.562
C05226=1203.816,140.869,-52.665,-178.255,6.035,148.563
C05227=1203.821,140.620,-52.645,-178.257,6.034,148.563
C05228=1203.826,140.371,-52.624,-178.260,6.032,148.564
C05229=1203.831,140.122,-52.604,-178.262,6.031,148.564
C05230=1203.836,139.872,-52.583,-178.265,6.030,148.564
C05231=1203.840,139.623,-52.563,-178.268,6.028,148.565
C05232=1203.845,139.374,-52.542,-178.270,6.027,148.565
C05233=1203.850,139.125,-52.521,-178.273,6.025,148.566
C05234=1203.854,138.876,-52.501,-178.276,6.024,148.566
C05235=1203.859,138.628,-52.481,-178.278,6.023,148.567
C05236=1203.864,138.379,-52.460,-178.281,6.021,148.567
C05237=1203.869,138.130,-52.439,-178.283,6.021,148.568
C05238=1203.873,137.881,-52.419,-178.286,6.019,148.568
C05239=1203.879,137.631,-52.399,-178.288,6.017,148.569
C05240=1203.883,137.382,-52.378,-178.291,6.016,148.569
C05241=1203.888,137.133,-52.358,-178.294,6.015,148.570
C05242=1203.893,136.884,-52.337,-178.296,6.014,148.570
C05243=1203.897,136.635,-52.317,-178.299,6.012,148.571
C05244=1203.902,136.385,-52.297,-178.301,6.011,148.571
C05245=1203.907,136.136,-52.276,-178.304,6.010,148.571
C05246=1203.912,135.887,-52.256,-178.307,6.008,148.572
C05247=1203.916,135.638,-52.235,-178.309,6.007,148.572
C05248=1203.920,135.389,-52.215,-178.312,6.005,148.573
C05249=1203.926,135.139,-52.195,-178.314,6.005,148.573
C05250=1203.930,134.890,-52.174,-178.317,6.003,148.574
C05251=1203.935,134.641,-52.154,-178.319,6.002,148.574
C05252=1203.940,134.393,-52.135,-178.322,6.001,148.575
C05253=1203.945,134.143,-52.114,-178.325,5.999,148.575
C05254=1203.950,133.894,-52.093,-178.327,5.998,148.576
C05255=1203.954,133.645,-52.073,-178.330,5.996,148.576
C05256=1203.960,133.376,-52.051,-178.333,5.995,148.577
C05257=1203.965,133.108,-52.030,-178.336,5.994,148.577
C05258=1203.970,132.839,-52.008,-178.338,5.992,148.578
C05259=1203.974,132.570,-51.986,-178.342,5.991,148.578
C05260=1203.980,132.322,-51.966,-178.344,5.990,148.579
C05261=1203.985,132.073,-51.945,-178.347,5.988,148.579
C05262=1203.989,131.823,-51.926,-178.349,5.987,148.580
C05263=1203.994,131.574,-51.905,-178.352,5.986,148.580
C05264=1203.999,131.324,-51.886,-178.355,5.984,148.581
C05265=1204.003,131.076,-51.865,-178.357,5.983,148.581
C05266=1204.008,130.826,-51.844,-178.360,5.982,148.581
C05267=1204.014,130.577,-51.825,-178.362,5.981,148.582
C05268=1204.018,130.328,-51.805,-178.365,5.979,148.582
C05269=1204.023,130.079,-51.785,-178.367,5.979,148.583
C05270=1204.027,129.830,-51.765,-178.370,5.977,148.583
C05271=1204.032,129.580,-51.745,-178.372,5.976,148.584
C05272=1204.037,129.332,-51.725,-178.375,5.974,148.584
C05273=1204.042,129.083,-51.705,-178.378,5.973,148.585
C05274=1204.046,128.834,-51.685,-178.380,5.972,148.585
C05275=1204.051,128.584,-51.665,-178.383,5.970,148.586
C05276=1204.056,128.335,-51.644,-178.386,5.969,148.586
C05277=1204.061,128.085,-51.625,-178.389,5.968,148.587
C05278=1204.066,127.837,-51.605,-178.391,5.967,148.587
C05279=1204.071,127.587,-51.585,-178.394,5.965,148.588
C05280=1204.075,127.338,-51.565,-178.396,5.965,148.588
C05281=1204.080,127.089,-51.545,-178.399,5.963,148.589
C05282=1204.085,126.840,-51.526,-178.401,5.962,148.589
C05283=1204.090,126.591,-51.505,-178.404,5.960,148.590
C05284=1204.094,126.341,-51.486,-178.406,5.959,148.590
C05285=1204.099,126.093,-51.465,-178.409,5.958,148.591
C05286=1204.103,125.843,-51.446,-178.412,5.957,148.591
C05287=1204.109,125.594,-51.426,-178.415,5.956,148.592
C05288=1204.113,125.345,-51.406,-178.417,5.955,148.592
C05289=1204.118,125.096,-51.386,-178.420,5.953,148.593
C05290=1204.123,124.846,-51.367,-178.422,5.952,148.593
C05291=1204.128,124.598,-51.347,-178.425,5.951,148.594
C05292=1204.132,124.348,-51.327,-178.427,5.950,148.594
C05293=1204.137,124.099,-51.307,-178.430,5.948,148.595
C05294=1204.142,123.850,-51.287,-178.432,5.947,148.595
C05295=1204.147,123.601,-51.268,-178.435,5.946,148.596
C05296=1204.151,123.352,-51.249,-178.438,5.945,148.596
C05297=1204.155,123.103,-51.228,-178.441,5.943,148.597
C05298=1204.161,122.854,-51.209,-178.443,5.942,148.597
C05299=1204.166,122.604,-51.189,-178.446,5.941,148.598
C05300=1204.170,122.355,-51.170,-178.448,5.940,148.598
C05301=1204.176,122.106,-51.150,-178.451,5.938,148.599
C05302=1204.180,121.857,-51.130,-178.453,5.938,148.599
C05303=1204.185,121.607,-51.110,-178.456,5.936,148.600
C05304=1204.190,121.358,-51.091,-178.459,5.935,148.600
C05305=1204.195,121.109,-51.071,-178.461,5.934,148.601
C05306=1204.199,120.860,-51.052,-178.464,5.933,148.601
C05307=1204.203,120.611,-51.032,-178.467,5.931,148.602
C05308=1204.209,120.362,-51.013,-178.469,5.930,148.602
C05309=1204.213,120.112,-50.993,-178.472,5.929,148.603
C05310=1204.219,119.863,-50.974,-178.474,5.928,148.603
C05311=1204.224,119.614,-50.954,-178.477,5.927,148.604
C05312=1204.228,119.364,-50.935,-178.479,5.926,148.604
C05313=1204.233,119.116,-50.916,-178.483,5.924,148.605
C05314=1204.237,118.867,-50.895,-178.485,5.923,148.605
C05315=1204.242,118.617,-50.876,-178.487,5.921,148.606
C05316=1204.247,118.368,-50.856,-178.490,5.921,148.606
C05317=1204.252,118.119,-50.837,-178.492,5.920,148.607
C05318=1204.256,117.869,-50.818,-178.495,5.918,148.607
C05319=1204.261,117.621,-50.798,-178.497,5.918,148.608
C05320=1204.266,117.371,-50.779,-178.501,5.916,148.608
C05321=1204.272,117.122,-50.760,-178.503,5.915,148.609
C05322=1204.276,116.873,-50.740,-178.506,5.914,148.609
C05323=1204.280,116.623,-50.721,-178.508,5.913,148.610
C05324=1204.286,116.374,-50.702,-178.511,5.911,148.610
C05325=1204.290,116.125,-50.682,-178.513,5.910,148.611
C05326=1204.295,115.876,-50.663,-178.516,5.909,148.611
C05327=1204.300,115.627,-50.644,-178.519,5.908,148.612
C05328=1204.304,115.377,-50.624,-178.521,5.906,148.612
C05329=1204.310,115.128,-50.605,-178.524,5.906,148.613
C05330=1204.314,114.879,-50.586,-178.526,5.905,148.613
C05331=1204.319,114.630,-50.566,-178.529,5.903,148.614
C05332=1204.324,114.381,-50.547,-178.531,5.902,148.614
C05333=1204.329,114.132,-50.528,-178.535,5.901,148.615
C05334=1204.333,113.882,-50.508,-178.537,5.900,148.615
C05335=1204.339,113.634,-50.489,-178.539,5.898,148.616
C05336=1204.344,113.383,-50.470,-178.542,5.898,148.616
C05337=1204.348,113.134,-50.451,-178.545,5.896,148.617
C05338=1204.353,112.885,-50.432,-178.547,5.895,148.617
C05339=1204.358,112.636,-50.412,-178.549,5.894,148.618
C05340=1204.362,112.387,-50.393,-178.553,5.893,148.618
C05341=1204.367,112.138,-50.374,-178.555,5.892,148.619
C05342=1204.372,111.889,-50.355,-178.558,5.891,148.619
C05343=1204.377,111.639,-50.336,-178.560,5.890,148.620
C05344=1204.382,111.390,-50.317,-178.563,5.888,148.621
C05345=1204.386,111.141,-50.298,-178.565,5.887,148.621
C05346=1204.391,110.892,-50.278,-178.568,5.887,148.622
C05347=1204.396,110.642,-50.259,-178.571,5.885,148.622
C05348=1204.401,110.393,-50.241,-178.573,5.884,148.623
C05349=1204.406,110.144,-50.221,-178.576,5.883,148.623
C05350=1204.410,109.895,-50.202,-178.579,5.882,148.624
C05351=1204.415,109.645,-50.183,-178.581,5.880,148.624
C05352=1204.420,109.396,-50.165,-178.584,5.880,148.625
C05353=1204.425,109.147,-50.145,-178.586,5.879,148.625
C05354=1204.429,108.898,-50.126,-178.589,5.877,148.626
C05355=1204.434,108.649,-50.107,-178.591,5.876,148.626
C05356=1204.440,108.399,-50.088,-178.595,5.875,148.627
C05357=1204.444,108.150,-50.069,-178.597,5.874,148.627
C05358=1204.449,107.901,-50.050,-178.599,5.873,148.628
C05359=1204.454,107.652,-50.032,-178.602,5.872,148.628
C05360=1204.459,107.383,-50.011,-178.605,5.871,148.629
C05361=1204.465,107.115,-49.991,-178.607,5.869,148.629
C05362=1204.469,106.846,-49.970,-178.610,5.868,148.630
C05363=1204.475,106.578,-49.950,-178.613,5.867,148.631
C05364=1204.479,106.329,-49.932,-178.616,5.866,148.631
C05365=1204.484,106.080,-49.912,-178.618,5.865,148.632
C05366=1204.489,105.830,-49.894,-178.621,5.864,148.632
C05367=1204.494,105.581,-49.874,-178.624,5.863,148.633
C05368=1204.499,105.332,-49.856,-178.626,5.862,148.633
C05369=1204.504,105.083,-49.837,-178.628,5.861,148.634
C05370=1204.508,104.833,-49.818,-178.631,5.859,148.634
C05371=1204.514,104.584,-49.799,-178.634,5.859,148.635
C05372=1204.518,104.335,-49.780,-178.636,5.857,148.635
C05373=1204.523,104.086,-49.762,-178.639,5.856,148.636
C05374=1204.528,103.837,-49.743,-178.642,5.856,148.636
C05375=1204.532,103.587,-49.725,-178.644,5.854,148.637
C05376=1204.538,103.338,-49.705,-178.647,5.854,148.638
C05377=1204.542,103.088,-49.687,-178.650,5.852,148.638
C05378=1204.547,102.839,-49.668,-178.652,5.851,148.639
C05379=1204.552,102.590,-49.650,-178.654,5.850,148.639
C05380=1204.556,102.341,-49.631,-178.658,5.849,148.640
C05381=1204.562,102.091,-49.612,-178.660,5.848,148.640
C05382=1204.566,101.843,-49.593,-178.662,5.847,148.641
C05383=1204.571,101.593,-49.575,-178.665,5.846,148.641
C05384=1204.576,101.343,-49.556,-178.668,5.845,148.642
C05385=1204.581,101.095,-49.538,-178.670,5.844,148.642
C05386=1204.585,100.845,-49.519,-178.673,5.843,148.643
C05387=1204.591,100.596,-49.500,-178.675,5.842,148.643
C05388=1204.596,100.347,-49.482,-178.678,5.840,148.644
C05389=1204.600,100.097,-49.464,-178.680,5.839,148.644
C05390=1204.605,99.848,-49.445,-178.683,5.839,148.645
C05391=1204.610,99.599,-49.427,-178.686,5.837,148.646
C05392=1204.614,99.350,-49.407,-178.688,5.836,148.646
C05393=1204.620,99.100,-49.389,-178.691,5.836,148.647
C05394=1204.625,98.851,-49.371,-178.694,5.834,148.647
C05395=1204.629,98.602,-49.352,-178.696,5.834,148.648
C05396=1204.634,98.353,-49.334,-178.698,5.833,148.648
C05397=1204.639,98.103,-49.315,-178.702,5.831,148.649
C05398=1204.644,97.854,-49.297,-178.704,5.830,148.649
C05399=1204.648,97.605,-49.278,-178.706,5.830,148.650
C05400=1204.654,97.355,-49.260,-178.709,5.828,148.650
C05401=1204.659,97.106,-49.242,-178.712,5.827,148.651
C05402=1204.663,96.857,-49.223,-178.714,5.827,148.652
C05403=1204.668,96.608,-49.205,-178.717,5.825,148.652
C05404=1204.673,96.358,-49.187,-178.720,5.824,148.653
C05405=1204.678,96.109,-49.168,-178.722,5.824,148.653
C05406=1204.683,95.860,-49.149,-178.725,5.822,148.654
C05407=1204.687,95.610,-49.131,-178.727,5.821,148.654
C05408=1204.692,95.361,-49.113,-178.730,5.821,148.655
C05409=1204.697,95.112,-49.095,-178.732,5.819,148.655
C05410=1204.703,94.863,-49.077,-178.735,5.818,148.656
C05411=1204.707,94.613,-49.058,-178.738,5.818,148.656
C05412=1204.712,94.364,-49.040,-178.740,5.816,148.657
C05413=1204.717,94.115,-49.022,-178.743,5.815,148.657
C05414=1204.721,93.866,-49.004,-178.745,5.814,148.658
C05415=1204.726,93.616,-48.985,-178.748,5.813,148.659
C05416=1204.731,93.366,-48.967,-178.750,5.812,148.659
C05417=1204.736,93.117,-48.949,-178.753,5.812,148.660
C05418=1204.741,92.869,-48.930,-178.756,5.810,148.660
C05419=1204.746,92.620,-48.912,-178.758,5.809,148.661
C05420=1204.750,92.370,-48.894,-178.761,5.809,148.661
C05421=1204.755,92.121,-48.876,-178.764,5.807,148.662
C05422=1204.760,91.871,-48.858,-178.766,5.806,148.662
C05423=1204.765,91.622,-48.840,-178.769,5.805,148.663
C05424=1204.771,91.373,-48.821,-178.772,5.804,148.663
C05425=1204.775,91.124,-48.803,-178.774,5.803,148.664
C05426=1204.780,90.874,-48.785,-178.776,5.802,148.665
C05427=1204.785,90.624,-48.767,-178.780,5.801,148.665
C05428=1204.790,90.375,-48.749,-178.782,5.800,148.666
C05429=1204.794,90.126,-48.731,-178.784,5.800,148.666
C05430=1204.799,89.877,-48.713,-178.787,5.799,148.667
C05431=1204.804,89.628,-48.695,-178.790,5.797,148.667
C05432=1204.809,89.378,-48.677,-178.792,5.797,148.668
C05433=1204.814,89.129,-48.659,-178.794,5.796,148.668
C05434=1204.818,88.880,-48.641,-178.798,5.794,148.669
C05435=1204.823,88.630,-48.623,-178.800,5.794,148.670
C05436=1204.828,88.381,-48.605,-178.802,5.793,148.670
C05437=1204.833,88.132,-48.587,-178.805,5.792,148.671
C05438=1204.838,87.883,-48.569,-178.808,5.791,148.671
C05439=1204.843,87.634,-48.551,-178.810,5.790,148.672
C05440=1204.847,87.384,-48.532,-178.813,5.789,148.672
C05441=1204.852,87.135,-48.514,-178.816,5.788,148.673
C05442=1204.857,86.885,-48.497,-178.818,5.787,148.674
C05443=1204.862,86.636,-48.479,-178.820,5.786,148.674
C05444=1204.867,86.386,-48.461,-178.823,5.786,148.675
C05445=1204.872,86.137,-48.443,-178.826,5.784,148.675
C05446=1204.877,85.888,-48.425,-178.828,5.783,148.676
C05447=1204.882,85.639,-48.407,-178.831,5.783,148.676
C05448=1204.887,85.390,-48.389,-178.834,5.781,148.677
C05449=1204.892,85.140,-48.372,-178.836,5.780,148.677
C05450=1204.897,84.891,-48.354,-178.839,5.780,148.678
C05451=1204.901,84.641,-48.336,-178.841,5.779,148.678
C05452=1204.906,84.392,-48.318,-178.844,5.778,148.679
C05453=1204.911,84.143,-48.300,-178.846,5.777,148.680
C05454=1204.916,83.893,-48.283,-178.849,5.776,148.680
C05455=1204.921,83.644,-48.265,-178.852,5.775,148.681
C05456=1204.925,83.395,-48.247,-178.854,5.774,148.681
C05457=1204.930,83.146,-48.229,-178.857,5.773,148.682
C05458=1204.936,82.896,-48.212,-178.859,5.772,148.682
C05459=1204.941,82.647,-48.194,-178.862,5.772,148.683
C05460=1204.945,82.397,-48.176,-178.865,5.770,148.684
C05461=1204.950,82.148,-48.158,-178.867,5.769,148.684
C05462=1204.955,81.899,-48.141,-178.870,5.769,148.685
C05463=1204.960,81.650,-48.123,-178.872,5.768,148.685
C05464=1204.965,81.381,-48.104,-178.875,5.766,148.686
C05465=1204.970,81.112,-48.085,-178.878,5.766,148.686
C05466=1204.975,80.844,-48.066,-178.881,5.764,148.687
C05467=1204.981,80.576,-48.047,-178.884,5.764,148.688
C05468=1204.986,80.327,-48.029,-178.886,5.763,148.688
C05469=1204.991,80.078,-48.011,-178.889,5.762,148.689
C05470=1204.996,79.828,-47.995,-178.892,5.761,148.689
C05471=1205.000,79.579,-47.977,-178.894,5.760,148.690
C05472=1205.006,79.329,-47.960,-178.896,5.760,148.691
C05473=1205.011,79.080,-47.942,-178.900,5.758,148.691
C05474=1205.016,78.831,-47.924,-178.902,5.757,148.692
